C01814=1073.013,225.555,417.556,174.109,27.687,154.920
C01815=1073.019,225.804,417.531,174.111,27.690,154.921
C01816=1073.025,226.052,417.504,174.113,27.694,154.921
C01817=1073.031,226.301,417.478,174.116,27.698,154.922
C01818=1073.036,226.549,417.451,174.118,27.702,154.923
C01819=1073.043,226.798,417.426,174.120,27.706,154.923
C01820=1073.048,227.046,417.399,174.123,27.710,154.924
C01821=1073.054,227.295,417.373,174.125,27.713,154.924
C01822=1073.060,227.544,417.348,174.127,27.717,154.925
C01823=1073.066,227.792,417.321,174.129,27.721,154.926
C01824=1073.072,228.041,417.295,174.131,27.725,154.926
C01825=1073.078,228.289,417.269,174.133,27.729,154.927
C01826=1073.084,228.538,417.243,174.136,27.733,154.927
C01827=1073.089,228.787,417.217,174.138,27.736,154.928
C01828=1073.096,229.036,417.190,174.140,27.740,154.929
C01829=1073.102,229.285,417.165,174.143,27.744,154.929
C01830=1073.107,229.533,417.138,174.145,27.748,154.930
C01831=1073.113,229.782,417.112,174.147,27.752,154.930
C01832=1073.119,230.030,417.086,174.150,27.755,154.931
C01833=1073.125,230.278,417.059,174.152,27.760,154.932
C01834=1073.131,230.527,417.033,174.154,27.764,154.932
C01835=1073.136,230.776,417.007,174.156,27.768,154.933
C01836=1073.142,231.024,416.980,174.158,27.771,154.933
C01837=1073.148,231.273,416.954,174.160,27.775,154.934
C01838=1073.153,231.521,416.927,174.163,27.779,154.935
C01839=1073.159,231.770,416.901,174.165,27.782,154.935
C01840=1073.165,232.018,416.874,174.167,27.787,154.936
C01841=1073.170,232.267,416.848,174.169,27.791,154.936
C01842=1073.177,232.515,416.822,174.172,27.795,154.937
C01843=1073.183,232.764,416.795,174.174,27.798,154.938
C01844=1073.189,233.013,416.769,174.176,27.802,154.938
C01845=1073.195,233.262,416.743,174.179,27.806,154.939
C01846=1073.200,233.510,416.716,174.181,27.810,154.939
C01847=1073.206,233.758,416.689,174.183,27.814,154.940
C01848=1073.212,234.007,416.663,174.186,27.818,154.941
C01849=1073.218,234.255,416.636,174.188,27.821,154.941
C01850=1073.223,234.504,416.610,174.190,27.825,154.942
C01851=1073.229,234.752,416.583,174.193,27.829,154.943
C01852=1073.235,235.001,416.557,174.195,27.833,154.943
C01853=1073.244,235.416,416.511,174.198,27.839,154.944
C01854=1073.254,235.831,416.467,174.202,27.846,154.945
C01855=1073.264,236.245,416.423,174.206,27.852,154.946
C01856=1073.273,236.660,416.377,174.210,27.859,154.947
C01857=1073.279,236.908,416.351,174.212,27.863,154.948
C01858=1073.285,237.157,416.324,174.214,27.867,154.948
C01859=1073.291,237.405,416.297,174.217,27.871,154.949
C01860=1073.296,237.653,416.271,174.219,27.874,154.950
C01861=1073.303,237.902,416.244,174.221,27.878,154.950
C01862=1073.309,238.151,416.217,174.224,27.882,154.951
C01863=1073.314,238.399,416.191,174.226,27.886,154.951
C01864=1073.320,238.648,416.164,174.228,27.890,154.952
C01865=1073.327,238.897,416.137,174.231,27.894,154.953
C01866=1073.332,239.145,416.110,174.233,27.897,154.953
C01867=1073.337,239.394,416.083,174.235,27.901,154.954
C01868=1073.343,239.642,416.056,174.238,27.905,154.954
C01869=1073.350,239.891,416.029,174.240,27.909,154.955
C01870=1073.355,240.139,416.003,174.242,27.913,154.956
C01871=1073.361,240.387,415.975,174.245,27.917,154.956
C01872=1073.367,240.636,415.949,174.247,27.920,154.957
C01873=1073.373,240.885,415.921,174.249,27.924,154.957
C01874=1073.379,241.133,415.894,174.252,27.928,154.958
C01875=1073.384,241.382,415.868,174.254,27.932,154.959
C01876=1073.390,241.629,415.840,174.257,27.936,154.959
C01877=1073.397,241.878,415.813,174.259,27.940,154.960
C01878=1073.402,242.127,415.786,174.261,27.943,154.960
C01879=1073.408,242.375,415.759,174.264,27.947,154.961
C01880=1073.414,242.624,415.732,174.266,27.951,154.962
C01881=1073.420,242.872,415.705,174.268,27.955,154.962
C01882=1073.425,243.121,415.678,174.271,27.959,154.963
C01883=1073.431,243.369,415.650,174.273,27.963,154.963
C01884=1073.438,243.618,415.623,174.275,27.967,154.964
C01885=1073.443,243.866,415.596,174.278,27.971,154.965
C01886=1073.449,244.114,415.569,174.280,27.975,154.965
C01887=1073.454,244.364,415.541,174.282,27.978,154.966
C01888=1073.460,244.612,415.515,174.285,27.982,154.966
C01889=1073.466,244.860,415.487,174.287,27.986,154.967
C01890=1073.472,245.109,415.460,174.289,27.990,154.968
C01891=1073.478,245.357,415.432,174.292,27.994,154.968
C01892=1073.483,245.605,415.405,174.294,27.998,154.969
C01893=1073.490,245.854,415.377,174.296,28.002,154.970
C01894=1073.495,246.103,415.350,174.300,28.005,154.970
C01895=1073.500,246.351,415.323,174.302,28.009,154.971
C01896=1073.507,246.599,415.296,174.304,28.013,154.971
C01897=1073.512,246.848,415.268,174.307,28.017,154.972
C01898=1073.518,247.096,415.241,174.309,28.021,154.972
C01899=1073.524,247.344,415.213,174.312,28.025,154.973
C01900=1073.529,247.593,415.185,174.314,28.029,154.974
C01901=1073.535,247.841,415.158,174.316,28.033,154.974
C01902=1073.541,248.090,415.131,174.319,28.036,154.975
C01903=1073.547,248.338,415.103,174.321,28.040,154.976
C01904=1073.552,248.587,415.076,174.323,28.045,154.976
C01905=1073.562,248.995,415.030,174.327,28.051,154.977
C01906=1073.571,249.403,414.985,174.331,28.057,154.978
C01907=1073.581,249.812,414.939,174.335,28.064,154.979
C01908=1073.590,250.219,414.893,174.339,28.070,154.980
C01909=1073.595,250.468,414.866,174.341,28.074,154.981
C01910=1073.601,250.716,414.839,174.344,28.078,154.982
C01911=1073.607,250.965,414.810,174.346,28.082,154.982
C01912=1073.613,251.213,414.782,174.348,28.086,154.983
C01913=1073.619,251.462,414.755,174.351,28.090,154.983
C01914=1073.624,251.710,414.727,174.353,28.094,154.984
C01915=1073.630,251.958,414.699,174.356,28.097,154.985
C01916=1073.636,252.206,414.672,174.359,28.101,154.985
C01917=1073.641,252.455,414.644,174.361,28.105,154.986
C01918=1073.647,252.704,414.616,174.363,28.109,154.986
C01919=1073.653,252.951,414.589,174.366,28.113,154.987
C01920=1073.659,253.200,414.560,174.368,28.117,154.988
C01921=1073.665,253.448,414.532,174.371,28.121,154.988
C01922=1073.671,253.697,414.505,174.373,28.125,154.989
C01923=1073.677,253.945,414.477,174.375,28.128,154.989
C01924=1073.683,254.193,414.448,174.378,28.132,154.990
C01925=1073.688,254.442,414.421,174.380,28.136,154.991
C01926=1073.694,254.691,414.393,174.383,28.140,154.991
C01927=1073.700,254.939,414.365,174.386,28.144,154.992
C01928=1073.706,255.187,414.337,174.388,28.148,154.993
C01929=1073.712,255.436,414.309,174.390,28.152,154.993
C01930=1073.718,255.684,414.281,174.393,28.156,154.994
C01931=1073.724,255.933,414.253,174.395,28.160,154.994
C01932=1073.729,256.181,414.225,174.398,28.164,154.995
C01933=1073.735,256.429,414.197,174.400,28.167,154.996
C01934=1073.741,256.677,414.169,174.402,28.171,154.996
C01935=1073.747,256.926,414.141,174.406,28.175,154.997
C01936=1073.753,257.175,414.113,174.408,28.179,154.997
C01937=1073.758,257.423,414.085,174.410,28.183,154.998
C01938=1073.765,257.671,414.056,174.413,28.187,154.999
C01939=1073.771,257.919,414.028,174.415,28.190,154.999
C01940=1073.776,258.167,414.000,174.418,28.194,155.000
C01941=1073.782,258.416,413.972,174.420,28.198,155.000
C01942=1073.788,258.664,413.944,174.422,28.202,155.001
C01943=1073.794,258.913,413.916,174.426,28.206,155.002
C01944=1073.800,259.161,413.888,174.428,28.210,155.002
C01945=1073.806,259.409,413.859,174.430,28.214,155.003
C01946=1073.812,259.657,413.831,174.433,28.217,155.003
C01947=1073.818,259.906,413.802,174.435,28.221,155.004
C01948=1073.824,260.154,413.775,174.438,28.225,155.005
C01949=1073.830,260.403,413.747,174.440,28.229,155.005
C01950=1073.836,260.651,413.718,174.443,28.233,155.006
C01951=1073.842,260.899,413.690,174.446,28.237,155.006
C01952=1073.847,261.148,413.661,174.448,28.241,155.007
C01953=1073.854,261.396,413.632,174.450,28.245,155.008
C01954=1073.860,261.644,413.605,174.453,28.248,155.008
C01955=1073.866,261.892,413.577,174.455,28.252,155.009
C01956=1073.872,262.140,413.548,174.459,28.256,155.009
C01957=1073.881,262.547,413.501,174.463,28.262,155.010
C01958=1073.891,262.952,413.455,174.467,28.268,155.011
C01959=1073.902,263.357,413.409,174.471,28.275,155.012
C01960=1073.911,263.764,413.362,174.475,28.281,155.013
C01961=1073.917,264.011,413.334,174.477,28.285,155.014
C01962=1073.923,264.260,413.305,174.480,28.289,155.015
C01963=1073.929,264.508,413.276,174.483,28.293,155.015
C01964=1073.934,264.756,413.248,174.485,28.297,155.016
C01965=1073.941,265.004,413.219,174.488,28.300,155.016
C01966=1073.946,265.253,413.190,174.490,28.304,155.017
C01967=1073.952,265.502,413.161,174.493,28.309,155.018
C01968=1073.957,265.750,413.133,174.496,28.312,155.018
C01969=1073.964,265.998,413.104,174.498,28.316,155.019
C01970=1073.970,266.246,413.075,174.500,28.320,155.019
C01971=1073.976,266.495,413.047,174.503,28.324,155.020
C01972=1073.981,266.742,413.018,174.505,28.328,155.021
C01973=1073.987,266.991,412.989,174.508,28.332,155.021
C01974=1073.993,267.239,412.960,174.511,28.336,155.022
C01975=1073.999,267.487,412.931,174.513,28.340,155.023
C01976=1074.005,267.736,412.903,174.516,28.343,155.023
C01977=1074.010,267.984,412.874,174.518,28.347,155.024
C01978=1074.016,268.232,412.845,174.521,28.352,155.025
C01979=1074.022,268.481,412.816,174.524,28.355,155.025
C01980=1074.028,268.729,412.787,174.526,28.359,155.026
C01981=1074.035,268.977,412.758,174.529,28.363,155.026
C01982=1074.040,269.226,412.728,174.532,28.367,155.027
C01983=1074.046,269.474,412.701,174.534,28.371,155.028
C01984=1074.052,269.722,412.671,174.537,28.375,155.028
C01985=1074.057,269.970,412.642,174.539,28.379,155.029
C01986=1074.064,270.218,412.613,174.542,28.383,155.029
C01987=1074.070,270.466,412.584,174.545,28.387,155.030
C01988=1074.076,270.715,412.555,174.547,28.391,155.031
C01989=1074.081,270.963,412.526,174.550,28.395,155.031
C01990=1074.087,271.211,412.497,174.552,28.399,155.032
C01991=1074.092,271.459,412.467,174.555,28.402,155.033
C01992=1074.099,271.708,412.438,174.558,28.406,155.033
C01993=1074.105,271.956,412.409,174.560,28.410,155.034
C01994=1074.110,272.204,412.380,174.563,28.414,155.034
C01995=1074.117,272.452,412.351,174.565,28.418,155.035
C01996=1074.123,272.700,412.322,174.568,28.423,155.036
C01997=1074.128,272.949,412.292,174.571,28.426,155.036
C01998=1074.134,273.196,412.263,174.573,28.430,155.037
C01999=1074.140,273.445,412.234,174.576,28.434,155.038
C02000=1074.146,273.693,412.205,174.579,28.438,155.038
C02001=1074.151,273.941,412.175,174.581,28.442,155.039
C02002=1074.158,274.189,412.146,174.584,28.446,155.040
C02003=1074.163,274.438,412.116,174.586,28.450,155.040
C02004=1074.169,274.686,412.087,174.589,28.454,155.041
C02005=1074.175,274.934,412.058,174.592,28.458,155.041
C02006=1074.181,275.183,412.029,174.594,28.462,155.042
C02007=1074.187,275.431,411.999,174.597,28.466,155.043
C02008=1074.193,275.679,411.970,174.600,28.470,155.043
C02009=1074.202,276.088,411.922,174.604,28.476,155.044
C02010=1074.212,276.496,411.872,174.609,28.483,155.045
C02011=1074.222,276.906,411.824,174.613,28.489,155.046
C02012=1074.232,277.314,411.776,174.617,28.496,155.047
C02013=1074.237,277.562,411.746,174.620,28.500,155.048
C02014=1074.243,277.811,411.717,174.623,28.504,155.049
C02015=1074.249,278.058,411.687,174.625,28.508,155.049
C02016=1074.255,278.307,411.657,174.627,28.512,155.050
C02017=1074.261,278.555,411.628,174.631,28.516,155.051
C02018=1074.267,278.803,411.598,174.633,28.520,155.051
C02019=1074.272,279.051,411.568,174.636,28.524,155.052
C02020=1074.279,279.299,411.539,174.639,28.528,155.052
C02021=1074.284,279.547,411.509,174.641,28.532,155.053
C02022=1074.290,279.796,411.479,174.644,28.536,155.054
C02023=1074.296,280.044,411.450,174.646,28.540,155.054
C02024=1074.303,280.292,411.419,174.650,28.544,155.055
C02025=1074.308,280.541,411.390,174.652,28.548,155.056
C02026=1074.315,280.788,411.360,174.654,28.552,155.056
C02027=1074.320,281.037,411.330,174.658,28.556,155.057
C02028=1074.326,281.285,411.301,174.660,28.560,155.058
C02029=1074.332,281.533,411.270,174.663,28.564,155.058
C02030=1074.337,281.781,411.241,174.666,28.568,155.059
C02031=1074.344,282.029,411.211,174.668,28.572,155.060
C02032=1074.349,282.277,411.181,174.671,28.576,155.060
C02033=1074.355,282.525,411.151,174.674,28.580,155.061
C02034=1074.361,282.773,411.121,174.676,28.584,155.062
C02035=1074.366,283.021,411.091,174.679,28.588,155.062
C02036=1074.372,283.269,411.061,174.681,28.592,155.063
C02037=1074.378,283.517,411.032,174.685,28.596,155.063
C02038=1074.385,283.766,411.001,174.687,28.600,155.064
C02039=1074.391,284.014,410.971,174.689,28.605,155.065
C02040=1074.396,284.262,410.941,174.693,28.609,155.066
C02041=1074.402,284.510,410.911,174.695,28.613,155.066
C02042=1074.407,284.758,410.881,174.698,28.617,155.067
C02043=1074.413,285.006,410.851,174.701,28.621,155.067
C02044=1074.419,285.254,410.820,174.703,28.625,155.068
C02045=1074.426,285.502,410.790,174.707,28.629,155.069
C02046=1074.432,285.751,410.760,174.709,28.633,155.069
C02047=1074.438,285.999,410.730,174.712,28.637,155.070
C02048=1074.443,286.246,410.700,174.715,28.641,155.071
C02049=1074.449,286.494,410.669,174.717,28.645,155.071
C02050=1074.455,286.743,410.639,174.720,28.649,155.072
C02051=1074.461,286.991,410.609,174.723,28.653,155.073
C02052=1074.467,287.239,410.579,174.726,28.657,155.073
C02053=1074.473,287.487,410.548,174.728,28.661,155.074
C02054=1074.479,287.735,410.518,174.731,28.665,155.075
C02055=1074.485,287.984,410.488,174.734,28.669,155.075
C02056=1074.491,288.231,410.458,174.736,28.673,155.076
C02057=1074.497,288.479,410.428,174.740,28.677,155.077
C02058=1074.503,288.727,410.398,174.742,28.681,155.077
C02059=1074.509,288.975,410.367,174.745,28.685,155.078
C02060=1074.515,289.223,410.336,174.748,28.689,155.078
C02061=1074.525,289.642,410.285,174.753,28.696,155.080
C02062=1074.535,290.061,410.234,174.757,28.703,155.081
C02063=1074.545,290.480,410.182,174.762,28.710,155.082
C02064=1074.555,290.899,410.131,174.767,28.717,155.083
C02065=1074.560,291.147,410.100,174.769,28.721,155.084
C02066=1074.566,291.396,410.069,174.772,28.725,155.084
C02067=1074.572,291.643,410.039,174.775,28.729,155.085
C02068=1074.578,291.891,410.008,174.777,28.734,155.086
C02069=1074.585,292.139,409.977,174.781,28.738,155.086
C02070=1074.591,292.387,409.947,174.783,28.742,155.087
C02071=1074.596,292.635,409.916,174.786,28.746,155.088
C02072=1074.602,292.883,409.885,174.789,28.750,155.088
C02073=1074.608,293.131,409.855,174.791,28.754,155.089
C02074=1074.614,293.379,409.824,174.795,28.758,155.090
C02075=1074.620,293.626,409.793,174.797,28.762,155.090
C02076=1074.626,293.875,409.762,174.800,28.766,155.091
C02077=1074.631,294.123,409.732,174.803,28.770,155.092
C02078=1074.638,294.372,409.701,174.806,28.775,155.092
C02079=1074.644,294.619,409.670,174.809,28.779,155.093
C02080=1074.650,294.867,409.639,174.811,28.783,155.094
C02081=1074.655,295.115,409.608,174.814,28.787,155.094
C02082=1074.662,295.363,409.577,174.817,28.792,155.095
C02083=1074.667,295.610,409.547,174.820,28.796,155.096
C02084=1074.673,295.859,409.515,174.823,28.800,155.096
C02085=1074.679,296.107,409.484,174.826,28.804,155.097
C02086=1074.686,296.355,409.454,174.828,28.808,155.098
C02087=1074.691,296.603,409.423,174.831,28.812,155.099
C02088=1074.697,296.850,409.392,174.834,28.816,155.099
C02089=1074.703,297.099,409.361,174.837,28.820,155.100
C02090=1074.709,297.346,409.329,174.840,28.825,155.101
C02091=1074.715,297.595,409.298,174.842,28.829,155.101
C02092=1074.720,297.842,409.267,174.846,28.833,155.102
C02093=1074.727,298.091,409.236,174.848,28.837,155.103
C02094=1074.732,298.339,409.204,174.852,28.842,155.103
C02095=1074.738,298.586,409.174,174.854,28.846,155.104
C02096=1074.744,298.835,409.142,174.857,28.850,155.105
C02097=1074.750,299.082,409.112,174.860,28.855,155.106
C02098=1074.755,299.330,409.080,174.862,28.858,155.106
C02099=1074.761,299.579,409.049,174.866,28.863,155.107
C02100=1074.767,299.826,409.018,174.868,28.867,155.108
C02101=1074.773,300.074,408.986,174.871,28.872,155.108
C02102=1074.779,300.322,408.955,174.874,28.876,155.109
C02103=1074.785,300.570,408.923,174.877,28.880,155.110
C02104=1074.790,300.818,408.892,174.880,28.884,155.110
C02105=1074.796,301.065,408.861,174.883,28.889,155.111
C02106=1074.802,301.314,408.829,174.885,28.893,155.112
C02107=1074.807,301.561,408.798,174.889,28.897,155.113
C02108=1074.814,301.810,408.767,174.891,28.901,155.113
C02109=1074.819,302.057,408.735,174.894,28.906,155.114
C02110=1074.825,302.305,408.703,174.897,28.910,155.115
C02111=1074.831,302.553,408.672,174.900,28.915,155.115
C02112=1074.837,302.801,408.640,174.903,28.918,155.116
C02113=1074.842,303.017,408.613,174.905,28.922,155.117
C02114=1074.847,303.235,408.585,174.908,28.926,155.117
C02115=1074.852,303.451,408.558,174.910,28.930,155.118
C02116=1074.858,303.668,408.530,174.913,28.934,155.119
C02117=1074.863,303.885,408.503,174.916,28.938,155.119
C02118=1074.868,304.102,408.475,174.919,28.941,155.120
C02119=1074.873,304.318,408.447,174.921,28.945,155.120
C02120=1074.879,304.535,408.420,174.923,28.949,155.121
C02121=1074.884,304.783,408.388,174.926,28.953,155.122
C02122=1074.890,305.031,408.356,174.929,28.957,155.123
C02123=1074.897,305.279,408.325,174.932,28.961,155.123
C02124=1074.902,305.526,408.293,174.935,28.966,155.124
C02125=1074.908,305.775,408.261,174.938,28.970,155.125
C02126=1074.914,306.022,408.230,174.941,28.975,155.125
C02127=1074.920,306.270,408.198,174.943,28.979,155.126
C02128=1074.926,306.518,408.166,174.947,28.983,155.127
C02129=1074.932,306.766,408.134,174.950,28.988,155.128
C02130=1074.938,307.014,408.103,174.952,28.992,155.128
C02131=1074.944,307.262,408.071,174.956,28.996,155.129
C02132=1074.950,307.509,408.039,174.958,29.000,155.130
C02133=1074.956,307.758,408.007,174.962,29.005,155.130
C02134=1074.962,308.005,407.976,174.964,29.009,155.131
C02135=1074.968,308.252,407.943,174.967,29.013,155.132
C02136=1074.974,308.501,407.911,174.970,29.018,155.133
C02137=1074.980,308.749,407.879,174.973,29.022,155.133
C02138=1074.986,308.996,407.848,174.977,29.027,155.134
C02139=1074.992,309.244,407.816,174.979,29.030,155.135
C02140=1074.998,309.492,407.784,174.982,29.035,155.136
C02141=1075.004,309.740,407.751,174.985,29.039,155.136
C02142=1075.011,309.987,407.720,174.988,29.044,155.137
C02143=1075.017,310.235,407.688,174.991,29.048,155.138
C02144=1075.023,310.484,407.656,174.994,29.052,155.138
C02145=1075.029,310.731,407.623,174.998,29.057,155.139
C02146=1075.035,310.979,407.591,175.000,29.061,155.140
C02147=1075.040,311.227,407.560,175.003,29.065,155.141
C02148=1075.047,311.474,407.528,175.006,29.070,155.141
C02149=1075.053,311.722,407.496,175.009,29.074,155.142
C02150=1075.059,311.971,407.464,175.013,29.078,155.143
C02151=1075.066,312.218,407.431,175.015,29.083,155.144
C02152=1075.072,312.466,407.399,175.018,29.087,155.144
C02153=1075.077,312.714,407.367,175.021,29.091,155.145
C02154=1075.084,312.961,407.335,175.024,29.096,155.146
C02155=1075.090,313.209,407.303,175.028,29.100,155.146
C02156=1075.096,313.457,407.270,175.030,29.104,155.147
C02157=1075.102,313.705,407.238,175.033,29.109,155.148
C02158=1075.109,313.953,407.205,175.036,29.113,155.149
C02159=1075.115,314.201,407.173,175.039,29.118,155.149
C02160=1075.121,314.449,407.141,175.043,29.122,155.150
C02161=1075.127,314.697,407.109,175.045,29.127,155.151
C02162=1075.132,314.944,407.076,175.048,29.131,155.152
C02163=1075.138,315.192,407.044,175.051,29.136,155.152
C02164=1075.144,315.440,407.011,175.054,29.140,155.153
C02165=1075.150,315.687,406.978,175.058,29.145,155.154
C02166=1075.156,315.936,406.946,175.060,29.149,155.155
C02167=1075.161,316.183,406.913,175.063,29.154,155.156
C02168=1075.168,316.431,406.880,175.066,29.158,155.156
C02169=1075.174,316.681,406.848,175.069,29.163,155.157
C02170=1075.180,316.930,406.815,175.073,29.168,155.158
C02171=1075.185,317.180,406.782,175.075,29.172,155.159
C02172=1075.191,317.429,406.750,175.078,29.177,155.159
C02173=1075.197,317.677,406.717,175.082,29.181,155.160
C02174=1075.203,317.925,406.683,175.084,29.186,155.161
C02175=1075.209,318.173,406.651,175.088,29.190,155.162
C02176=1075.215,318.420,406.618,175.091,29.195,155.163
C02177=1075.221,318.669,406.585,175.093,29.199,155.163
C02178=1075.227,318.916,406.553,175.097,29.204,155.164
C02179=1075.233,319.164,406.520,175.100,29.209,155.165
C02180=1075.239,319.412,406.487,175.103,29.213,155.166
C02181=1075.245,319.659,406.454,175.106,29.218,155.167
C02182=1075.251,319.907,406.420,175.108,29.222,155.167
C02183=1075.257,320.155,406.388,175.112,29.227,155.168
C02184=1075.263,320.403,406.356,175.115,29.232,155.169
C02185=1075.268,320.651,406.322,175.118,29.236,155.170
C02186=1075.275,320.899,406.290,175.121,29.241,155.170
C02187=1075.280,321.146,406.256,175.124,29.246,155.171
C02188=1075.287,321.394,406.224,175.127,29.250,155.172
C02189=1075.292,321.611,406.195,175.130,29.254,155.173
C02190=1075.297,321.829,406.165,175.133,29.258,155.173
C02191=1075.302,322.046,406.137,175.135,29.262,155.174
C02192=1075.308,322.263,406.107,175.138,29.266,155.175
C02193=1075.313,322.480,406.079,175.141,29.270,155.175
C02194=1075.318,322.698,406.049,175.144,29.274,155.176
C02195=1075.324,322.916,406.020,175.146,29.279,155.177
C02196=1075.329,323.133,405.991,175.149,29.282,155.178
C02197=1075.335,323.380,405.959,175.152,29.287,155.178
C02198=1075.341,323.628,405.925,175.155,29.292,155.179
C02199=1075.347,323.876,405.893,175.158,29.297,155.180
C02200=1075.353,324.125,405.859,175.161,29.301,155.181
C02201=1075.360,324.372,405.825,175.165,29.306,155.182
C02202=1075.365,324.619,405.792,175.168,29.310,155.182
C02203=1075.371,324.867,405.759,175.170,29.315,155.183
C02204=1075.377,325.115,405.726,175.174,29.320,155.184
C02205=1075.383,325.363,405.693,175.177,29.324,155.185
C02206=1075.390,325.611,405.659,175.180,29.329,155.186
C02207=1075.396,325.858,405.626,175.183,29.334,155.187
C02208=1075.402,326.106,405.593,175.186,29.339,155.187
C02209=1075.408,326.353,405.559,175.190,29.343,155.188
C02210=1075.414,326.601,405.526,175.192,29.347,155.189
C02211=1075.421,326.849,405.493,175.196,29.353,155.190
C02212=1075.426,327.096,405.459,175.199,29.357,155.191
C02213=1075.433,327.344,405.426,175.202,29.362,155.191
C02214=1075.438,327.592,405.393,175.205,29.367,155.192
C02215=1075.446,327.840,405.359,175.208,29.371,155.193
C02216=1075.451,328.088,405.325,175.212,29.376,155.194
C02217=1075.458,328.335,405.292,175.215,29.381,155.195
C02218=1075.463,328.582,405.259,175.217,29.385,155.195
C02219=1075.470,328.830,405.224,175.221,29.390,155.196
C02220=1075.476,329.078,405.192,175.224,29.395,155.197
C02221=1075.482,329.325,405.157,175.228,29.400,155.198
C02222=1075.489,329.574,405.124,175.231,29.404,155.199
C02223=1075.495,329.821,405.090,175.233,29.409,155.200
C02224=1075.501,330.068,405.058,175.237,29.414,155.200
C02225=1075.506,330.283,405.028,175.239,29.418,155.201
C02226=1075.512,330.500,404.999,175.243,29.422,155.202
C02227=1075.518,330.714,404.969,175.245,29.426,155.203
C02228=1075.522,330.930,404.940,175.248,29.430,155.203
C02229=1075.528,331.145,404.911,175.251,29.434,155.204
C02230=1075.534,331.359,404.882,175.254,29.439,155.205
C02231=1075.538,331.575,404.852,175.256,29.443,155.206
C02232=1075.543,331.790,404.822,175.259,29.447,155.206
C02233=1075.551,332.038,404.789,175.262,29.452,155.207
C02234=1075.556,332.286,404.755,175.265,29.457,155.208
C02235=1075.562,332.533,404.721,175.269,29.462,155.209
C02236=1075.568,332.781,404.687,175.272,29.467,155.210
C02237=1075.574,333.028,404.653,175.275,29.472,155.211
C02238=1075.580,333.276,404.619,175.278,29.476,155.211
C02239=1075.586,333.524,404.585,175.281,29.481,155.212
C02240=1075.592,333.771,404.551,175.285,29.486,155.213
C02241=1075.598,334.019,404.517,175.288,29.491,155.214
C02242=1075.605,334.267,404.482,175.292,29.496,155.215
C02243=1075.610,334.514,404.448,175.294,29.501,155.216
C02244=1075.616,334.761,404.414,175.297,29.506,155.217
C02245=1075.622,335.010,404.381,175.301,29.511,155.218
C02246=1075.628,335.257,404.347,175.304,29.516,155.218
C02247=1075.635,335.505,404.313,175.308,29.521,155.219
C02248=1075.641,335.752,404.279,175.311,29.526,155.220
C02249=1075.648,336.000,404.244,175.313,29.531,155.221
C02250=1075.654,336.247,404.210,175.317,29.536,155.222
C02251=1075.660,336.495,404.176,175.320,29.541,155.223
C02252=1075.666,336.743,404.142,175.324,29.546,155.224
C02253=1075.672,336.991,404.107,175.327,29.550,155.224
C02254=1075.679,337.237,404.073,175.330,29.556,155.225
C02255=1075.685,337.485,404.038,175.334,29.561,155.226
C02256=1075.691,337.732,404.004,175.336,29.565,155.227
C02257=1075.697,337.980,403.970,175.340,29.571,155.228
C02258=1075.703,338.228,403.935,175.343,29.576,155.229
C02259=1075.708,338.475,403.901,175.346,29.581,155.230
C02260=1075.715,338.723,403.867,175.350,29.586,155.231
C02261=1075.721,338.970,403.832,175.353,29.591,155.232
C02262=1075.727,339.218,403.797,175.357,29.596,155.233
C02263=1075.733,339.466,403.763,175.360,29.601,155.233
C02264=1075.739,339.714,403.728,175.362,29.606,155.234
C02265=1075.745,339.960,403.694,175.366,29.611,155.235
C02266=1075.752,340.208,403.659,175.369,29.616,155.236
C02267=1075.758,340.456,403.625,175.373,29.622,155.237
C02268=1075.764,340.703,403.589,175.376,29.627,155.238
C02269=1075.770,340.951,403.555,175.379,29.632,155.239
C02270=1075.776,341.198,403.521,175.383,29.637,155.240
C02271=1075.783,341.446,403.486,175.386,29.642,155.241
C02272=1075.788,341.693,403.451,175.390,29.647,155.242
C02273=1075.795,341.941,403.416,175.393,29.652,155.243
C02274=1075.801,342.189,403.382,175.396,29.658,155.244
C02275=1075.807,342.436,403.348,175.399,29.662,155.245
C02276=1075.813,342.684,403.312,175.402,29.668,155.246
C02277=1075.819,342.932,403.277,175.406,29.673,155.247
C02278=1075.826,343.178,403.243,175.409,29.678,155.247
C02279=1075.832,343.426,403.208,175.412,29.683,155.248
C02280=1075.838,343.674,403.172,175.416,29.689,155.249
C02281=1075.843,343.886,403.142,175.419,29.693,155.250
C02282=1075.849,344.099,403.113,175.422,29.698,155.251
C02283=1075.854,344.311,403.083,175.424,29.702,155.252
C02284=1075.859,344.524,403.053,175.428,29.706,155.253
C02285=1075.865,344.736,403.022,175.430,29.711,155.253
C02286=1075.869,344.949,402.993,175.434,29.716,155.254
C02287=1075.875,345.162,402.963,175.436,29.720,155.255
C02288=1075.880,345.374,402.933,175.439,29.724,155.256
C02289=1075.886,345.621,402.897,175.442,29.730,155.257
C02290=1075.893,345.869,402.863,175.445,29.735,155.258
C02291=1075.899,346.116,402.828,175.449,29.741,155.259
C02292=1075.905,346.364,402.792,175.452,29.746,155.260
C02293=1075.912,346.611,402.757,175.456,29.751,155.261
C02294=1075.917,346.858,402.722,175.459,29.757,155.262
C02295=1075.923,347.106,402.687,175.462,29.762,155.263
C02296=1075.930,347.354,402.651,175.466,29.767,155.264
C02297=1075.936,347.601,402.616,175.469,29.772,155.265
C02298=1075.942,347.848,402.581,175.473,29.778,155.266
C02299=1075.948,348.096,402.545,175.476,29.783,155.267
C02300=1075.955,348.343,402.510,175.479,29.789,155.268
C02301=1075.961,348.591,402.474,175.483,29.794,155.269
C02302=1075.968,348.838,402.439,175.486,29.800,155.270
C02303=1075.973,349.085,402.404,175.490,29.805,155.270
C02304=1075.979,349.333,402.368,175.493,29.810,155.272
C02305=1075.986,349.580,402.333,175.496,29.816,155.273
C02306=1075.992,349.828,402.297,175.500,29.821,155.274
C02307=1075.999,350.075,402.262,175.503,29.826,155.274
C02308=1076.004,350.322,402.227,175.507,29.832,155.276
C02309=1076.010,350.570,402.191,175.510,29.837,155.277
C02310=1076.017,350.817,402.156,175.513,29.843,155.278
C02311=1076.023,351.065,402.120,175.517,29.849,155.279
C02312=1076.030,351.312,402.085,175.520,29.854,155.280
C02313=1076.036,351.560,402.049,175.524,29.859,155.281
C02314=1076.042,351.807,402.013,175.528,29.865,155.282
C02315=1076.048,352.054,401.978,175.531,29.870,155.283
C02316=1076.054,352.301,401.942,175.535,29.876,155.284
C02317=1076.060,352.549,401.907,175.538,29.881,155.285
C02318=1076.066,352.797,401.871,175.542,29.887,155.286
C02319=1076.073,353.043,401.835,175.545,29.893,155.287
C02320=1076.079,353.291,401.799,175.548,29.898,155.288
C02321=1076.085,353.539,401.764,175.552,29.904,155.289
C02322=1076.092,353.786,401.727,175.555,29.909,155.290
C02323=1076.098,354.033,401.691,175.559,29.915,155.291
C02324=1076.104,354.281,401.656,175.562,29.921,155.292
C02325=1076.110,354.527,401.620,175.565,29.926,155.293
C02326=1076.116,354.775,401.584,175.569,29.932,155.294
C02327=1076.123,355.022,401.548,175.572,29.937,155.295
C02328=1076.129,355.270,401.512,175.576,29.943,155.296
C02329=1076.135,355.517,401.476,175.580,29.949,155.297
C02330=1076.141,355.764,401.440,175.583,29.955,155.298
C02331=1076.147,356.011,401.404,175.587,29.960,155.299
C02332=1076.153,356.259,401.368,175.590,29.966,155.300
C02333=1076.160,356.506,401.332,175.593,29.972,155.302
C02334=1076.166,356.753,401.296,175.597,29.977,155.303
C02335=1076.173,357.001,401.260,175.600,29.983,155.304
C02336=1076.179,357.248,401.223,175.604,29.989,155.305
C02337=1076.185,357.463,401.192,175.607,29.994,155.306
C02338=1076.190,357.677,401.161,175.611,29.999,155.307
C02339=1076.195,357.891,401.129,175.613,30.004,155.307
C02340=1076.201,358.105,401.099,175.617,30.009,155.308
C02341=1076.207,358.319,401.067,175.619,30.013,155.309
C02342=1076.212,358.534,401.035,175.623,30.018,155.310
C02343=1076.217,358.747,401.004,175.626,30.024,155.311
C02344=1076.223,358.962,400.973,175.628,30.029,155.312
C02345=1076.230,359.209,400.936,175.632,30.034,155.313
C02346=1076.236,359.457,400.900,175.635,30.040,155.314
C02347=1076.242,359.704,400.863,175.640,30.046,155.315
C02348=1076.248,359.951,400.828,175.643,30.052,155.317
C02349=1076.255,360.198,400.791,175.646,30.058,155.318
C02350=1076.260,360.446,400.754,175.650,30.063,155.319
C02351=1076.267,360.693,400.718,175.653,30.070,155.320
C02352=1076.273,360.940,400.681,175.657,30.076,155.321
C02353=1076.279,361.187,400.645,175.661,30.081,155.322
C02354=1076.286,361.434,400.608,175.664,30.087,155.323
C02355=1076.293,361.682,400.571,175.668,30.093,155.324
C02356=1076.299,361.929,400.535,175.671,30.099,155.326
C02357=1076.305,362.176,400.499,175.675,30.105,155.327
C02358=1076.311,362.423,400.462,175.679,30.111,155.328
C02359=1076.317,362.670,400.425,175.682,30.117,155.329
C02360=1076.324,362.918,400.388,175.686,30.123,155.330
C02361=1076.330,363.165,400.352,175.689,30.129,155.331
C02362=1076.337,363.412,400.315,175.693,30.135,155.332
C02363=1076.343,363.659,400.278,175.697,30.141,155.334
C02364=1076.349,363.906,400.241,175.700,30.147,155.335
C02365=1076.356,364.154,400.204,175.704,30.153,155.336
C02366=1076.362,364.401,400.168,175.707,30.159,155.337
C02367=1076.369,364.648,400.131,175.711,30.165,155.338
C02368=1076.375,364.894,400.094,175.715,30.172,155.339
C02369=1076.381,365.142,400.057,175.718,30.178,155.341
C02370=1076.388,365.389,400.020,175.722,30.184,155.342
C02371=1076.393,365.637,399.983,175.725,30.190,155.343
C02372=1076.400,365.883,399.946,175.730,30.196,155.344
C02373=1076.406,366.131,399.909,175.733,30.202,155.345
C02374=1076.413,366.378,399.872,175.736,30.208,155.346
C02375=1076.418,366.625,399.835,175.740,30.214,155.348
C02376=1076.425,366.872,399.798,175.744,30.220,155.349
C02377=1076.432,367.119,399.761,175.748,30.227,155.350
C02378=1076.438,367.366,399.724,175.751,30.233,155.351
C02379=1076.444,367.613,399.687,175.754,30.239,155.352
C02380=1076.451,367.861,399.649,175.759,30.246,155.354
C02381=1076.457,368.107,399.612,175.762,30.252,155.355
C02382=1076.463,368.355,399.575,175.766,30.258,155.356
C02383=1076.470,368.602,399.537,175.769,30.264,155.357
C02384=1076.476,368.849,399.500,175.773,30.271,155.359
C02385=1076.482,369.096,399.463,175.777,30.277,155.360
C02386=1076.489,369.343,399.425,175.780,30.283,155.361
C02387=1076.495,369.590,399.389,175.785,30.289,155.362
C02388=1076.501,369.837,399.351,175.788,30.296,155.363
C02389=1076.508,370.084,399.313,175.791,30.302,155.365
C02390=1076.514,370.331,399.276,175.796,30.309,155.366
C02391=1076.521,370.579,399.239,175.799,30.315,155.367
C02392=1076.527,370.825,399.201,175.803,30.321,155.368
C02393=1076.533,371.048,399.168,175.806,30.327,155.369
C02394=1076.538,371.270,399.133,175.810,30.333,155.371
C02395=1076.545,371.493,399.100,175.813,30.338,155.372
C02396=1076.551,371.715,399.066,175.816,30.344,155.373
C02397=1076.556,371.937,399.032,175.820,30.350,155.374
C02398=1076.562,372.160,398.999,175.823,30.356,155.375
C02399=1076.568,372.383,398.964,175.827,30.362,155.376
C02400=1076.574,372.605,398.931,175.829,30.368,155.377
C02401=1076.580,372.852,398.893,175.834,30.374,155.379
C02402=1076.587,373.099,398.855,175.837,30.380,155.380
C02403=1076.594,373.346,398.817,175.842,30.387,155.381
C02404=1076.600,373.593,398.780,175.845,30.393,155.382
C02405=1076.607,373.840,398.742,175.848,30.400,155.384
C02406=1076.613,374.087,398.704,175.853,30.407,155.385
C02407=1076.619,374.334,398.666,175.856,30.413,155.386
C02408=1076.625,374.581,398.628,175.860,30.420,155.388
C02409=1076.632,374.828,398.590,175.864,30.427,155.389
C02410=1076.639,375.074,398.552,175.867,30.433,155.390
C02411=1076.645,375.322,398.514,175.871,30.440,155.392
C02412=1076.651,375.569,398.477,175.875,30.447,155.393
C02413=1076.657,375.816,398.438,175.879,30.453,155.394
C02414=1076.663,376.063,398.401,175.883,30.460,155.396
C02415=1076.670,376.310,398.362,175.886,30.467,155.397
C02416=1076.677,376.556,398.325,175.890,30.473,155.398
C02417=1076.683,376.804,398.287,175.894,30.480,155.400
C02418=1076.690,377.050,398.248,175.898,30.487,155.401
C02419=1076.696,377.297,398.210,175.902,30.494,155.402
C02420=1076.703,377.545,398.172,175.906,30.501,155.404
C02421=1076.709,377.791,398.133,175.910,30.507,155.405
C02422=1076.715,378.038,398.095,175.913,30.514,155.406
C02423=1076.722,378.285,398.056,175.917,30.521,155.408
C02424=1076.729,378.532,398.018,175.921,30.528,155.409
C02425=1076.736,378.778,397.980,175.925,30.535,155.410
C02426=1076.742,379.026,397.942,175.929,30.541,155.412
C02427=1076.749,379.272,397.903,175.932,30.548,155.413
C02428=1076.755,379.519,397.866,175.937,30.555,155.415
C02429=1076.762,379.766,397.827,175.940,30.562,155.416
C02430=1076.768,380.014,397.789,175.945,30.569,155.417
C02431=1076.775,380.260,397.750,175.948,30.576,155.419
C02432=1076.781,380.507,397.712,175.952,30.583,155.420
C02433=1076.788,380.754,397.673,175.956,30.590,155.421
C02434=1076.794,381.001,397.634,175.960,30.597,155.423
C02435=1076.801,381.248,397.596,175.964,30.604,155.424
C02436=1076.807,381.494,397.558,175.968,30.611,155.426
C02437=1076.814,381.741,397.519,175.972,30.618,155.427
C02438=1076.821,381.988,397.480,175.976,30.625,155.428
C02439=1076.827,382.235,397.442,175.979,30.632,155.430
C02440=1076.834,382.482,397.403,175.984,30.639,155.431
C02441=1076.840,382.729,397.364,175.987,30.646,155.433
C02442=1076.846,382.975,397.325,175.992,30.653,155.434
C02443=1076.853,383.222,397.287,175.995,30.660,155.436
C02444=1076.860,383.469,397.248,176.000,30.668,155.437
C02445=1076.867,383.716,397.209,176.003,30.675,155.439
C02446=1076.872,383.962,397.170,176.007,30.682,155.440
C02447=1076.879,384.209,397.131,176.011,30.690,155.442
C02448=1076.886,384.456,397.092,176.015,30.697,155.443
C02449=1076.892,384.693,397.054,176.019,30.704,155.444
C02450=1076.898,384.930,397.017,176.023,30.711,155.446
C02451=1076.905,385.167,396.980,176.027,30.718,155.447
C02452=1076.910,385.404,396.942,176.030,30.725,155.449
C02453=1076.918,385.641,396.905,176.034,30.732,155.450
C02454=1076.923,385.878,396.867,176.038,30.739,155.451
C02455=1076.930,386.115,396.830,176.042,30.746,155.453
C02456=1076.936,386.351,396.792,176.046,30.753,155.454
C02457=1076.943,386.598,396.753,176.049,30.760,155.456
C02458=1076.950,386.845,396.714,176.054,30.768,155.457
C02459=1076.956,387.092,396.675,176.058,30.775,155.459
C02460=1076.963,387.338,396.635,176.062,30.782,155.460
C02461=1076.970,387.585,396.596,176.066,30.790,155.462
C02462=1076.976,387.832,396.557,176.070,30.797,155.463
C02463=1076.983,388.078,396.517,176.074,30.805,155.465
C02464=1076.990,388.325,396.479,176.078,30.812,155.466
C02465=1076.996,388.572,396.439,176.082,30.820,155.468
C02466=1077.003,388.819,396.400,176.086,30.827,155.470
C02467=1077.010,389.065,396.361,176.091,30.835,155.471
C02468=1077.016,389.312,396.321,176.094,30.842,155.473
C02469=1077.023,389.559,396.282,176.098,30.850,155.474
C02470=1077.029,389.805,396.242,176.103,30.858,155.476
C02471=1077.037,390.053,396.202,176.106,30.865,155.477
C02472=1077.044,390.299,396.163,176.111,30.873,155.479
C02473=1077.050,390.546,396.123,176.115,30.880,155.480
C02474=1077.057,390.792,396.084,176.119,30.888,155.482
C02475=1077.063,391.039,396.044,176.123,30.896,155.484
C02476=1077.070,391.286,396.005,176.128,30.903,155.485
C02477=1077.077,391.532,395.965,176.131,30.911,155.487
C02478=1077.084,391.778,395.925,176.135,30.919,155.488
C02479=1077.090,392.026,395.885,176.140,30.927,155.490
C02480=1077.097,392.272,395.846,176.144,30.934,155.492
C02481=1077.104,392.519,395.806,176.148,30.942,155.493
C02482=1077.110,392.765,395.765,176.152,30.950,155.495
C02483=1077.117,393.012,395.726,176.157,30.958,155.496
C02484=1077.124,393.259,395.686,176.160,30.966,155.498
C02485=1077.130,393.506,395.646,176.165,30.974,155.500
C02486=1077.137,393.752,395.606,176.169,30.982,155.501
C02487=1077.144,393.999,395.566,176.174,30.989,155.503
C02488=1077.150,394.245,395.526,176.177,30.997,155.505
C02489=1077.158,394.492,395.486,176.181,31.005,155.506
C02490=1077.164,394.739,395.446,176.186,31.013,155.508
C02491=1077.171,394.985,395.406,176.190,31.022,155.510
C02492=1077.178,395.232,395.365,176.194,31.029,155.511
C02493=1077.185,395.479,395.326,176.198,31.037,155.513
C02494=1077.191,395.725,395.286,176.203,31.046,155.515
C02495=1077.197,395.972,395.246,176.207,31.054,155.516
C02496=1077.205,396.218,395.204,176.211,31.062,155.518
C02497=1077.211,396.465,395.164,176.215,31.070,155.520
C02498=1077.218,396.711,395.124,176.220,31.079,155.522
C02499=1077.225,396.958,395.084,176.224,31.087,155.523
C02500=1077.232,397.205,395.044,176.229,31.095,155.525
C02501=1077.239,397.451,395.003,176.232,31.103,155.527
C02502=1077.245,397.698,394.963,176.237,31.111,155.528
C02503=1077.252,397.944,394.922,176.241,31.120,155.530
C02504=1077.259,398.191,394.881,176.245,31.128,155.532
C02505=1077.266,398.436,394.841,176.250,31.136,155.534
C02506=1077.272,398.679,394.801,176.253,31.144,155.535
C02507=1077.279,398.924,394.761,176.258,31.153,155.537
C02508=1077.286,399.168,394.721,176.262,31.161,155.539
C02509=1077.293,399.412,394.681,176.267,31.169,155.541
C02510=1077.300,399.657,394.640,176.271,31.178,155.542
C02511=1077.307,399.901,394.600,176.275,31.186,155.544
C02512=1077.312,400.145,394.560,176.279,31.194,155.546
C02513=1077.320,400.392,394.518,176.284,31.203,155.548
C02514=1077.326,400.638,394.478,176.288,31.212,155.550
C02515=1077.333,400.885,394.437,176.293,31.220,155.551
C02516=1077.340,401.131,394.396,176.297,31.229,155.553
C02517=1077.347,401.378,394.356,176.302,31.237,155.555
C02518=1077.354,401.625,394.314,176.305,31.245,155.557
C02519=1077.361,401.871,394.274,176.310,31.254,155.559
C02520=1077.368,402.117,394.232,176.314,31.263,155.561
C02521=1077.375,402.364,394.192,176.319,31.271,155.562
C02522=1077.381,402.611,394.150,176.323,31.280,155.564
C02523=1077.388,402.857,394.109,176.328,31.289,155.566
C02524=1077.395,403.103,394.068,176.332,31.298,155.568
C02525=1077.402,403.350,394.027,176.337,31.306,155.570
C02526=1077.410,403.596,393.986,176.341,31.315,155.572
C02527=1077.416,403.843,393.946,176.346,31.324,155.574
C02528=1077.423,404.090,393.904,176.350,31.333,155.576
C02529=1077.430,404.336,393.863,176.355,31.342,155.577
C02530=1077.437,404.583,393.821,176.359,31.351,155.579
C02531=1077.444,404.829,393.781,176.364,31.360,155.581
C02532=1077.450,405.076,393.739,176.368,31.368,155.583
C02533=1077.458,405.322,393.697,176.373,31.377,155.585
C02534=1077.465,405.568,393.656,176.377,31.387,155.587
C02535=1077.471,405.815,393.614,176.382,31.396,155.589
C02536=1077.479,406.061,393.573,176.386,31.405,155.591
C02537=1077.485,406.308,393.531,176.391,31.414,155.593
C02538=1077.492,406.555,393.490,176.395,31.423,155.595
C02539=1077.499,406.800,393.448,176.400,31.432,155.597
C02540=1077.506,407.047,393.406,176.405,31.441,155.599
C02541=1077.513,407.293,393.365,176.409,31.450,155.601
C02542=1077.520,407.540,393.323,176.414,31.460,155.603
C02543=1077.527,407.786,393.281,176.418,31.469,155.605
C02544=1077.534,408.033,393.240,176.423,31.478,155.607
C02545=1077.541,408.278,393.198,176.427,31.488,155.609
C02546=1077.547,408.525,393.156,176.433,31.497,155.611
C02547=1077.554,408.772,393.114,176.437,31.506,155.613
C02548=1077.562,409.018,393.072,176.442,31.516,155.615
C02549=1077.568,409.265,393.030,176.446,31.525,155.617
C02550=1077.576,409.511,392.989,176.451,31.535,155.619
C02551=1077.583,409.757,392.946,176.455,31.544,155.621
C02552=1077.590,410.003,392.904,176.460,31.553,155.623
C02553=1077.597,410.250,392.862,176.465,31.563,155.625
C02554=1077.604,410.497,392.820,176.470,31.573,155.627
C02555=1077.611,410.743,392.778,176.475,31.582,155.629
C02556=1077.618,410.989,392.736,176.479,31.591,155.631
C02557=1077.625,411.236,392.693,176.484,31.601,155.634
C02558=1077.632,411.482,392.652,176.488,31.611,155.636
C02559=1077.639,411.728,392.609,176.494,31.620,155.638
C02560=1077.647,411.974,392.567,176.499,31.630,155.640
C02561=1077.653,412.220,392.525,176.503,31.640,155.642
C02562=1077.660,412.465,392.483,176.508,31.650,155.644
C02563=1077.667,412.711,392.441,176.513,31.659,155.646
C02564=1077.675,412.956,392.398,176.518,31.669,155.648
C02565=1077.682,413.202,392.357,176.522,31.679,155.650
C02566=1077.688,413.448,392.314,176.527,31.689,155.653
C02567=1077.696,413.693,392.272,176.533,31.699,155.655
C02568=1077.703,413.939,392.230,176.537,31.709,155.657
C02569=1077.710,414.185,392.187,176.542,31.718,155.659
C02570=1077.717,414.430,392.144,176.546,31.728,155.661
C02571=1077.724,414.677,392.101,176.552,31.738,155.663
C02572=1077.732,414.923,392.059,176.557,31.748,155.666
C02573=1077.739,415.170,392.017,176.561,31.758,155.668
C02574=1077.746,415.416,391.974,176.567,31.768,155.670
C02575=1077.753,415.662,391.931,176.571,31.778,155.672
C02576=1077.761,415.909,391.888,176.576,31.789,155.675
C02577=1077.768,416.155,391.845,176.582,31.799,155.677
C02578=1077.775,416.401,391.802,176.586,31.809,155.679
C02579=1077.782,416.647,391.760,176.592,31.819,155.681
C02580=1077.789,416.893,391.716,176.597,31.829,155.684
C02581=1077.796,417.140,391.673,176.601,31.840,155.686
C02582=1077.803,417.385,391.630,176.607,31.850,155.688
C02583=1077.810,417.632,391.588,176.612,31.860,155.691
C02584=1077.818,417.878,391.544,176.617,31.871,155.693
C02585=1077.825,418.124,391.501,176.622,31.881,155.695
C02586=1077.832,418.370,391.458,176.626,31.891,155.697
C02587=1077.840,418.616,391.415,176.632,31.902,155.700
C02588=1077.847,418.862,391.372,176.637,31.913,155.702
C02589=1077.854,419.109,391.328,176.642,31.923,155.705
C02590=1077.862,419.355,391.285,176.647,31.934,155.707
C02591=1077.868,419.601,391.243,176.653,31.945,155.709
C02592=1077.876,419.847,391.199,176.657,31.955,155.712
C02593=1077.883,420.093,391.156,176.663,31.966,155.714
C02594=1077.891,420.339,391.112,176.668,31.976,155.716
C02595=1077.898,420.585,391.069,176.673,31.987,155.719
C02596=1077.906,420.831,391.025,176.678,31.998,155.721
C02597=1077.912,421.077,390.981,176.684,32.009,155.724
C02598=1077.920,421.324,390.938,176.689,32.020,155.726
C02599=1077.927,421.569,390.894,176.694,32.031,155.729
C02600=1077.935,421.816,390.851,176.700,32.042,155.731
C02601=1077.942,422.061,390.808,176.705,32.052,155.733
C02602=1077.949,422.308,390.763,176.710,32.063,155.736
C02603=1077.957,422.554,390.720,176.715,32.074,155.738
C02604=1077.964,422.800,390.676,176.721,32.086,155.741
C02605=1077.971,423.045,390.632,176.726,32.097,155.743
C02606=1077.979,423.292,390.588,176.731,32.107,155.746
C02607=1077.987,423.538,390.545,176.737,32.119,155.748
C02608=1077.993,423.783,390.500,176.743,32.130,155.751
C02609=1078.001,424.030,390.457,176.747,32.141,155.754
C02610=1078.007,424.276,390.413,176.753,32.153,155.756
C02611=1078.016,424.521,390.368,176.759,32.164,155.759
C02612=1078.023,424.768,390.325,176.764,32.175,155.761
C02613=1078.030,425.013,390.280,176.769,32.186,155.764
C02614=1078.038,425.260,390.237,176.775,32.198,155.766
C02615=1078.045,425.506,390.192,176.780,32.209,155.769
C02616=1078.053,425.751,390.147,176.786,32.221,155.772
C02617=1078.061,426.013,390.101,176.791,32.233,155.774
C02618=1078.069,426.276,390.053,176.797,32.245,155.777
C02619=1078.077,426.538,390.006,176.804,32.258,155.780
C02620=1078.085,426.799,389.959,176.810,32.270,155.783
C02621=1078.092,427.046,389.915,176.815,32.282,155.785
C02622=1078.100,427.292,389.870,176.820,32.293,155.788
C02623=1078.108,427.538,389.826,176.826,32.305,155.791
C02624=1078.115,427.784,389.781,176.832,32.317,155.793
C02625=1078.123,428.029,389.737,176.838,32.329,155.796
C02626=1078.130,428.275,389.692,176.843,32.341,155.799
C02627=1078.138,428.521,389.647,176.848,32.352,155.802
C02628=1078.145,428.767,389.603,176.854,32.364,155.804
C02629=1078.153,429.013,389.558,176.860,32.376,155.807
C02630=1078.161,429.258,389.513,176.866,32.388,155.810
C02631=1078.168,429.504,389.468,176.872,32.400,155.813
C02632=1078.175,429.750,389.423,176.877,32.412,155.815
C02633=1078.182,429.996,389.379,176.883,32.424,155.818
C02634=1078.190,430.241,389.334,176.889,32.437,155.821
C02635=1078.198,430.487,389.289,176.895,32.449,155.824
C02636=1078.205,430.733,389.244,176.900,32.461,155.827
C02637=1078.213,430.978,389.199,176.906,32.473,155.829
C02638=1078.221,431.224,389.154,176.912,32.486,155.832
C02639=1078.228,431.470,389.109,176.917,32.498,155.835
C02640=1078.236,431.716,389.063,176.923,32.510,155.838
C02641=1078.244,431.962,389.019,176.929,32.523,155.841
C02642=1078.252,432.208,388.973,176.935,32.535,155.844
C02643=1078.259,432.454,388.928,176.941,32.548,155.847
C02644=1078.267,432.699,388.882,176.947,32.560,155.849
C02645=1078.275,432.945,388.837,176.953,32.573,155.852
C02646=1078.282,433.191,388.792,176.959,32.586,155.855
C02647=1078.290,433.436,388.746,176.965,32.598,155.858
C02648=1078.297,433.681,388.701,176.971,32.611,155.861
C02649=1078.305,433.927,388.655,176.978,32.624,155.864
C02650=1078.313,434.172,388.609,176.984,32.637,155.867
C02651=1078.321,434.419,388.564,176.989,32.649,155.870
C02652=1078.328,434.665,388.518,176.995,32.663,155.873
C02653=1078.336,434.910,388.473,177.001,32.675,155.876
C02654=1078.343,435.155,388.427,177.007,32.688,155.879
C02655=1078.351,435.401,388.381,177.013,32.701,155.882
C02656=1078.359,435.647,388.335,177.019,32.714,155.885
C02657=1078.367,435.892,388.290,177.025,32.727,155.889
C02658=1078.375,436.137,388.243,177.032,32.741,155.892
C02659=1078.383,436.383,388.198,177.038,32.754,155.895
C02660=1078.391,436.629,388.152,177.044,32.767,155.898
C02661=1078.398,436.874,388.106,177.050,32.780,155.901
C02662=1078.406,437.120,388.060,177.056,32.794,155.904
C02663=1078.414,437.365,388.013,177.063,32.807,155.907
C02664=1078.422,437.611,387.967,177.070,32.820,155.910
C02665=1078.430,437.857,387.921,177.076,32.834,155.913
C02666=1078.438,438.102,387.875,177.083,32.847,155.917
C02667=1078.445,438.347,387.829,177.089,32.861,155.920
C02668=1078.454,438.593,387.783,177.095,32.874,155.923
C02669=1078.462,438.838,387.737,177.101,32.888,155.926
C02670=1078.470,439.084,387.690,177.108,32.902,155.930
C02671=1078.478,439.330,387.643,177.114,32.915,155.933
C02672=1078.486,439.575,387.597,177.120,32.929,155.936
C02673=1078.497,439.941,387.528,177.130,32.950,155.941
C02674=1078.510,440.308,387.458,177.140,32.970,155.946
C02675=1078.521,440.674,387.388,177.150,32.992,155.951
C02676=1078.533,441.039,387.319,177.160,33.013,155.956
C02677=1078.542,441.285,387.272,177.166,33.027,155.959
C02678=1078.549,441.531,387.225,177.172,33.041,155.963
C02679=1078.557,441.776,387.178,177.180,33.055,155.966
C02680=1078.565,442.021,387.131,177.186,33.069,155.969
C02681=1078.574,442.267,387.084,177.193,33.084,155.973
C02682=1078.581,442.512,387.037,177.199,33.098,155.976
C02683=1078.589,442.758,386.991,177.206,33.113,155.980
C02684=1078.597,443.003,386.943,177.213,33.127,155.983
C02685=1078.606,443.248,386.896,177.220,33.141,155.987
C02686=1078.613,443.493,386.849,177.226,33.156,155.990
C02687=1078.622,443.739,386.802,177.233,33.171,155.994
C02688=1078.630,443.984,386.754,177.241,33.185,155.997
C02689=1078.639,444.230,386.707,177.247,33.200,156.001
C02690=1078.646,444.474,386.660,177.254,33.215,156.004
C02691=1078.655,444.720,386.613,177.261,33.230,156.008
C02692=1078.663,444.965,386.565,177.268,33.244,156.011
C02693=1078.670,445.211,386.518,177.275,33.260,156.015
C02694=1078.679,445.456,386.470,177.282,33.275,156.019
C02695=1078.687,445.701,386.422,177.289,33.290,156.022
C02696=1078.696,445.946,386.374,177.296,33.305,156.026
C02697=1078.704,446.191,386.327,177.303,33.320,156.030
C02698=1078.712,446.436,386.280,177.310,33.335,156.033
C02699=1078.720,446.681,386.232,177.316,33.350,156.037
C02700=1078.728,446.926,386.184,177.323,33.365,156.041
C02701=1078.737,447.171,386.136,177.328,33.381,156.045
C02702=1078.745,447.416,386.088,177.335,33.396,156.048
C02703=1078.754,447.662,386.040,177.340,33.411,156.052
C02704=1078.762,447.908,385.992,177.346,33.426,156.056
C02705=1078.771,448.152,385.944,177.350,33.441,156.059
C02706=1078.779,448.398,385.896,177.355,33.456,156.063
C02707=1078.787,448.643,385.848,177.360,33.471,156.067
C02708=1078.795,448.887,385.799,177.364,33.486,156.071
C02709=1078.805,449.132,385.752,177.368,33.501,156.074
C02710=1078.815,449.377,385.705,177.373,33.515,156.078
C02711=1078.827,449.623,385.659,177.376,33.528,156.081
C02712=1078.841,449.869,385.614,177.381,33.541,156.085
C02713=1078.478,449.864,385.387,177.357,33.704,156.128
C02714=1078.459,449.535,385.447,177.351,33.687,156.123
C02715=1078.444,449.207,385.509,177.345,33.669,156.119
C02716=1078.431,448.882,385.573,177.340,33.649,156.114
C02717=1078.420,448.556,385.637,177.334,33.629,156.109
C02718=1078.412,448.311,385.685,177.329,33.614,156.105
C02719=1078.403,448.066,385.732,177.324,33.599,156.102
C02720=1078.395,447.821,385.780,177.318,33.584,156.098
C02721=1078.387,447.575,385.828,177.313,33.569,156.094
C02722=1078.379,447.330,385.876,177.307,33.554,156.090
C02723=1078.371,447.086,385.925,177.302,33.539,156.087
C02724=1078.362,446.841,385.973,177.295,33.523,156.083
C02725=1078.354,446.595,386.021,177.288,33.508,156.079
C02726=1078.346,446.350,386.068,177.282,33.493,156.075
C02727=1078.337,446.105,386.115,177.275,33.478,156.072
C02728=1078.329,445.860,386.164,177.267,33.463,156.068
C02729=1078.321,445.614,386.212,177.261,33.448,156.064
C02730=1078.313,445.369,386.260,177.253,33.433,156.061
C02731=1078.304,445.124,386.307,177.246,33.418,156.057
C02732=1078.296,444.878,386.354,177.239,33.403,156.053
C02733=1078.288,444.633,386.402,177.232,33.388,156.050
C02734=1078.279,444.388,386.450,177.224,33.373,156.046
C02735=1078.271,444.143,386.497,177.218,33.359,156.043
C02736=1078.263,443.898,386.544,177.211,33.343,156.039
C02737=1078.255,443.653,386.592,177.204,33.329,156.036
C02738=1078.246,443.408,386.639,177.197,33.315,156.032
C02739=1078.239,443.162,386.686,177.190,33.300,156.029
C02740=1078.230,442.916,386.733,177.183,33.285,156.025
C02741=1078.222,442.672,386.781,177.176,33.271,156.022
C02742=1078.214,442.426,386.827,177.170,33.256,156.018
C02743=1078.206,442.180,386.875,177.162,33.242,156.015
C02744=1078.198,441.936,386.921,177.156,33.228,156.011
C02745=1078.190,441.690,386.968,177.150,33.213,156.008
C02746=1078.181,441.445,387.016,177.142,33.199,156.004
C02747=1078.173,441.199,387.063,177.136,33.185,156.001
C02748=1078.166,440.954,387.110,177.129,33.171,155.998
C02749=1078.157,440.709,387.156,177.123,33.157,155.994
C02750=1078.149,440.441,387.207,177.115,33.142,155.991
C02751=1078.140,440.173,387.258,177.108,33.127,155.987
C02752=1078.131,439.906,387.309,177.101,33.111,155.983
C02753=1078.123,439.637,387.360,177.094,33.096,155.980
C02754=1078.115,439.392,387.406,177.087,33.082,155.977
C02755=1078.107,439.146,387.452,177.080,33.069,155.973
C02756=1078.099,438.901,387.499,177.074,33.055,155.970
C02757=1078.091,438.656,387.546,177.068,33.041,155.967
C02758=1078.083,438.410,387.592,177.061,33.028,155.964
C02759=1078.075,438.165,387.638,177.055,33.014,155.960
C02760=1078.066,437.919,387.684,177.048,33.001,155.957
C02761=1078.058,437.674,387.731,177.042,32.987,155.954
C02762=1078.051,437.428,387.777,177.035,32.974,155.951
C02763=1078.042,437.183,387.823,177.029,32.961,155.948
C02764=1078.035,436.937,387.869,177.023,32.947,155.944
C02765=1078.027,436.691,387.915,177.017,32.934,155.941
C02766=1078.019,436.446,387.962,177.010,32.920,155.938
C02767=1078.011,436.201,388.008,177.004,32.908,155.935
C02768=1078.003,435.955,388.054,176.997,32.894,155.932
C02769=1077.996,435.709,388.099,176.991,32.881,155.929
C02770=1077.988,435.464,388.145,176.985,32.868,155.926
C02771=1077.980,435.218,388.191,176.979,32.855,155.923
C02772=1077.972,434.972,388.236,176.972,32.842,155.920
C02773=1077.964,434.727,388.282,176.966,32.829,155.917
C02774=1077.957,434.481,388.328,176.960,32.816,155.914
C02775=1077.949,434.236,388.373,176.954,32.803,155.911
C02776=1077.941,433.990,388.419,176.948,32.791,155.908
C02777=1077.933,433.744,388.465,176.942,32.778,155.905
C02778=1077.926,433.499,388.511,176.936,32.765,155.902
C02779=1077.918,433.253,388.556,176.930,32.752,155.899
C02780=1077.910,433.008,388.602,176.924,32.740,155.896
C02781=1077.903,432.762,388.647,176.918,32.727,155.893
C02782=1077.895,432.517,388.693,176.912,32.714,155.890
C02783=1077.888,432.271,388.738,176.906,32.702,155.887
C02784=1077.880,432.024,388.784,176.900,32.689,155.884
C02785=1077.871,431.779,388.829,176.894,32.677,155.881
C02786=1077.864,431.533,388.874,176.888,32.665,155.878
C02787=1077.857,431.288,388.919,176.882,32.652,155.876
C02788=1077.849,431.042,388.964,176.876,32.640,155.873
C02789=1077.841,430.797,389.009,176.870,32.628,155.870
C02790=1077.833,430.550,389.054,176.864,32.615,155.867
C02791=1077.826,430.304,389.099,176.858,32.603,155.864
C02792=1077.819,430.059,389.145,176.852,32.591,155.861
C02793=1077.810,429.813,389.189,176.846,32.579,155.859
C02794=1077.803,429.567,389.234,176.840,32.567,155.856
C02795=1077.796,429.321,389.279,176.835,32.555,155.853
C02796=1077.787,429.076,389.324,176.830,32.543,155.850
C02797=1077.780,428.830,389.369,176.824,32.530,155.847
C02798=1077.773,428.584,389.414,176.818,32.519,155.845
C02799=1077.765,428.339,389.458,176.812,32.507,155.842
C02800=1077.758,428.093,389.503,176.806,32.495,155.839
C02801=1077.751,427.847,389.548,176.801,32.483,155.837
C02802=1077.743,427.601,389.592,176.795,32.471,155.834
C02803=1077.735,427.355,389.637,176.789,32.460,155.831
C02804=1077.727,427.109,389.681,176.783,32.448,155.829
C02805=1077.720,426.863,389.726,176.778,32.437,155.826
C02806=1077.711,426.600,389.773,176.772,32.424,155.823
C02807=1077.704,426.336,389.821,176.766,32.412,155.820
C02808=1077.696,426.073,389.868,176.760,32.399,155.817
C02809=1077.688,425.809,389.916,176.754,32.387,155.815
C02810=1077.680,425.563,389.960,176.748,32.376,155.812
C02811=1077.673,425.317,390.004,176.743,32.364,155.809
C02812=1077.665,425.071,390.049,176.738,32.353,155.807
C02813=1077.657,424.825,390.092,176.732,32.341,155.804
C02814=1077.650,424.579,390.137,176.726,32.330,155.802
C02815=1077.642,424.333,390.180,176.720,32.319,155.799
C02816=1077.636,424.087,390.225,176.716,32.307,155.796
C02817=1077.628,423.841,390.269,176.710,32.296,155.794
C02818=1077.620,423.595,390.313,176.705,32.285,155.791
C02819=1077.613,423.349,390.357,176.699,32.274,155.789
C02820=1077.606,423.103,390.400,176.693,32.263,155.786
C02821=1077.598,422.858,390.444,176.689,32.251,155.784
C02822=1077.591,422.611,390.489,176.683,32.240,155.781
C02823=1077.583,422.365,390.532,176.677,32.229,155.779
C02824=1077.576,422.119,390.576,176.672,32.218,155.776
C02825=1077.569,421.873,390.620,176.666,32.207,155.774
C02826=1077.562,421.627,390.664,176.662,32.196,155.771
C02827=1077.554,421.381,390.707,176.656,32.185,155.769
C02828=1077.547,421.135,390.751,176.651,32.175,155.766
C02829=1077.540,420.889,390.795,176.645,32.164,155.764
C02830=1077.533,420.643,390.838,176.641,32.153,155.762
C02831=1077.525,420.397,390.882,176.635,32.142,155.759
C02832=1077.518,420.151,390.925,176.629,32.132,155.757
C02833=1077.510,419.905,390.969,176.624,32.121,155.754
C02834=1077.503,419.659,391.012,176.619,32.110,155.752
C02835=1077.495,419.412,391.055,176.614,32.100,155.750
C02836=1077.488,419.166,391.098,176.609,32.089,155.747
C02837=1077.480,418.920,391.142,176.603,32.079,155.745
C02838=1077.473,418.674,391.185,176.599,32.068,155.743
C02839=1077.466,418.427,391.228,176.593,32.057,155.740
C02840=1077.459,418.182,391.271,176.588,32.047,155.738
C02841=1077.451,417.936,391.314,176.583,32.037,155.736
C02842=1077.444,417.689,391.357,176.578,32.026,155.733
C02843=1077.437,417.443,391.400,176.572,32.016,155.731
C02844=1077.430,417.198,391.444,176.568,32.005,155.729
C02845=1077.422,416.951,391.487,176.563,31.995,155.726
C02846=1077.415,416.705,391.530,176.557,31.985,155.724
C02847=1077.408,416.459,391.572,176.552,31.975,155.722
C02848=1077.401,416.213,391.616,176.548,31.965,155.720
C02849=1077.394,415.966,391.659,176.542,31.954,155.717
C02850=1077.387,415.720,391.701,176.537,31.944,155.715
C02851=1077.380,415.474,391.744,176.533,31.934,155.713
C02852=1077.373,415.228,391.787,176.527,31.924,155.711
C02853=1077.365,414.981,391.830,176.522,31.914,155.708
C02854=1077.358,414.735,391.873,176.518,31.903,155.706
C02855=1077.350,414.489,391.915,176.512,31.893,155.704
C02856=1077.344,414.243,391.958,176.507,31.884,155.702
C02857=1077.336,413.996,392.000,176.503,31.874,155.699
C02858=1077.329,413.750,392.043,176.497,31.864,155.697
C02859=1077.322,413.504,392.085,176.492,31.854,155.695
C02860=1077.315,413.257,392.127,176.488,31.844,155.693
C02861=1077.308,413.012,392.171,176.483,31.834,155.691
C02862=1077.300,412.766,392.213,176.477,31.825,155.689
C02863=1077.293,412.520,392.255,176.473,31.815,155.687
C02864=1077.285,412.273,392.297,176.468,31.805,155.684
C02865=1077.279,412.026,392.339,176.464,31.796,155.682
C02866=1077.272,411.780,392.382,176.458,31.785,155.680
C02867=1077.264,411.534,392.424,176.453,31.776,155.678
C02868=1077.257,411.287,392.466,176.449,31.767,155.676
C02869=1077.250,411.041,392.509,176.444,31.757,155.674
C02870=1077.243,410.795,392.551,176.439,31.747,155.672
C02871=1077.236,410.548,392.593,176.434,31.738,155.670
C02872=1077.229,410.302,392.635,176.429,31.728,155.668
C02873=1077.222,410.056,392.677,176.425,31.719,155.665
C02874=1077.215,409.810,392.720,176.420,31.709,155.663
C02875=1077.208,409.563,392.761,176.415,31.700,155.661
C02876=1077.201,409.317,392.803,176.411,31.691,155.659
C02877=1077.194,409.070,392.845,176.406,31.681,155.657
C02878=1077.187,408.824,392.887,176.400,31.671,155.655
C02879=1077.180,408.577,392.929,176.396,31.662,155.653
C02880=1077.173,408.332,392.971,176.391,31.653,155.651
C02881=1077.167,408.085,393.012,176.387,31.643,155.649
C02882=1077.159,407.839,393.054,176.382,31.634,155.647
C02883=1077.152,407.592,393.096,176.377,31.625,155.645
C02884=1077.145,407.346,393.138,176.373,31.616,155.643
C02885=1077.138,407.099,393.180,176.368,31.606,155.641
C02886=1077.131,406.853,393.221,176.364,31.597,155.639
C02887=1077.125,406.607,393.263,176.359,31.588,155.637
C02888=1077.117,406.360,393.305,176.355,31.579,155.635
C02889=1077.111,406.113,393.346,176.350,31.570,155.633
C02890=1077.104,405.867,393.388,176.345,31.561,155.631
C02891=1077.096,405.621,393.430,176.341,31.552,155.629
C02892=1077.090,405.375,393.471,176.336,31.542,155.627
C02893=1077.083,405.128,393.512,176.332,31.534,155.625
C02894=1077.075,404.881,393.554,176.327,31.525,155.623
C02895=1077.069,404.635,393.595,176.323,31.516,155.621
C02896=1077.062,404.389,393.636,176.318,31.507,155.620
C02897=1077.055,404.142,393.677,176.313,31.498,155.618
C02898=1077.048,403.895,393.719,176.309,31.489,155.616
C02899=1077.041,403.649,393.760,176.304,31.480,155.614
C02900=1077.034,403.403,393.801,176.300,31.472,155.612
C02901=1077.027,403.156,393.843,176.295,31.463,155.610
C02902=1077.020,402.910,393.884,176.291,31.454,155.608
C02903=1077.013,402.664,393.925,176.286,31.445,155.606
C02904=1077.007,402.417,393.966,176.281,31.437,155.605
C02905=1076.999,402.170,394.008,176.277,31.428,155.603
C02906=1076.993,401.924,394.048,176.272,31.419,155.601
C02907=1076.986,401.677,394.089,176.269,31.411,155.599
C02908=1076.978,401.430,394.130,176.264,31.402,155.597
C02909=1076.972,401.185,394.171,176.260,31.393,155.595
C02910=1076.965,400.937,394.212,176.255,31.385,155.593
C02911=1076.958,400.691,394.253,176.251,31.376,155.592
C02912=1076.951,400.445,394.294,176.246,31.368,155.590
C02913=1076.945,400.198,394.335,176.242,31.359,155.588
C02914=1076.937,399.953,394.376,176.237,31.351,155.586
C02915=1076.930,399.708,394.415,176.233,31.342,155.584
C02916=1076.924,399.463,394.456,176.229,31.334,155.583
C02917=1076.917,399.219,394.497,176.224,31.325,155.581
C02918=1076.911,398.973,394.537,176.220,31.317,155.579
C02919=1076.904,398.728,394.577,176.215,31.309,155.577
C02920=1076.897,398.483,394.617,176.212,31.301,155.576
C02921=1076.891,398.239,394.658,176.207,31.293,155.574
C02922=1076.883,397.992,394.698,176.203,31.284,155.572
C02923=1076.876,397.745,394.738,176.198,31.275,155.570
C02924=1076.869,397.499,394.780,176.194,31.267,155.569
C02925=1076.863,397.252,394.820,176.190,31.259,155.567
C02926=1076.856,397.005,394.860,176.186,31.251,155.565
C02927=1076.849,396.758,394.901,176.181,31.243,155.563
C02928=1076.843,396.512,394.941,176.177,31.234,155.562
C02929=1076.836,396.265,394.982,176.173,31.227,155.560
C02930=1076.829,396.019,395.021,176.169,31.219,155.558
C02931=1076.822,395.773,395.062,176.164,31.210,155.557
C02932=1076.815,395.525,395.102,176.160,31.202,155.555
C02933=1076.809,395.279,395.143,176.156,31.194,155.553
C02934=1076.802,395.033,395.183,176.152,31.186,155.551
C02935=1076.794,394.786,395.223,176.147,31.178,155.550
C02936=1076.788,394.539,395.263,176.143,31.170,155.548
C02937=1076.782,394.293,395.303,176.139,31.162,155.546
C02938=1076.775,394.046,395.343,176.135,31.154,155.545
C02939=1076.768,393.800,395.383,176.130,31.146,155.543
C02940=1076.761,393.553,395.424,176.126,31.138,155.541
C02941=1076.755,393.307,395.464,176.122,31.130,155.540
C02942=1076.748,393.060,395.503,176.118,31.122,155.538
C02943=1076.741,392.812,395.543,176.113,31.114,155.537
C02944=1076.735,392.566,395.583,176.110,31.107,155.535
C02945=1076.728,392.320,395.623,176.105,31.098,155.533
C02946=1076.721,392.073,395.663,176.101,31.091,155.532
C02947=1076.714,391.827,395.702,176.097,31.083,155.530
C02948=1076.707,391.579,395.742,176.093,31.075,155.528
C02949=1076.701,391.333,395.782,176.088,31.067,155.527
C02950=1076.694,391.087,395.822,176.085,31.060,155.525
C02951=1076.688,390.839,395.861,176.080,31.052,155.524
C02952=1076.681,390.593,395.901,176.076,31.044,155.522
C02953=1076.674,390.347,395.940,176.072,31.037,155.520
C02954=1076.667,390.099,395.980,176.068,31.029,155.519
C02955=1076.660,389.853,396.020,176.063,31.022,155.517
C02956=1076.654,389.606,396.059,176.060,31.014,155.516
C02957=1076.647,389.360,396.099,176.055,31.006,155.514
C02958=1076.639,389.113,396.138,176.051,30.999,155.513
C02959=1076.633,388.866,396.178,176.047,30.991,155.511
C02960=1076.627,388.619,396.217,176.043,30.984,155.510
C02961=1076.619,388.373,396.256,176.038,30.976,155.508
C02962=1076.613,388.126,396.296,176.035,30.969,155.506
C02963=1076.606,387.880,396.335,176.030,30.961,155.505
C02964=1076.599,387.633,396.374,176.027,30.954,155.503
C02965=1076.593,387.386,396.413,176.022,30.947,155.502
C02966=1076.586,387.140,396.453,176.018,30.939,155.500
C02967=1076.579,386.893,396.492,176.014,30.932,155.499
C02968=1076.573,386.646,396.531,176.010,30.924,155.497
C02969=1076.566,386.400,396.571,176.006,30.917,155.496
C02970=1076.560,386.161,396.608,176.002,30.910,155.494
C02971=1076.554,385.923,396.646,175.998,30.903,155.493
C02972=1076.547,385.686,396.684,175.994,30.896,155.492
C02973=1076.541,385.449,396.721,175.990,30.889,155.490
C02974=1076.535,385.211,396.759,175.987,30.882,155.489
C02975=1076.528,384.973,396.796,175.982,30.875,155.487
C02976=1076.522,384.736,396.834,175.979,30.868,155.486
C02977=1076.516,384.498,396.872,175.975,30.860,155.484
C02978=1076.509,384.251,396.911,175.971,30.853,155.483
C02979=1076.503,384.005,396.949,175.967,30.846,155.481
C02980=1076.496,383.759,396.988,175.963,30.839,155.480
C02981=1076.490,383.511,397.028,175.959,30.832,155.479
C02982=1076.483,383.265,397.066,175.955,30.824,155.477
C02983=1076.476,383.018,397.105,175.951,30.817,155.476
C02984=1076.469,382.771,397.144,175.947,30.810,155.474
C02985=1076.464,382.525,397.183,175.943,30.803,155.473
C02986=1076.457,382.278,397.222,175.939,30.796,155.471
C02987=1076.450,382.031,397.261,175.935,30.788,155.470
C02988=1076.444,381.783,397.299,175.931,30.782,155.468
C02989=1076.437,381.537,397.337,175.927,30.774,155.467
C02990=1076.431,381.290,397.376,175.923,30.767,155.466
C02991=1076.424,381.044,397.415,175.919,30.760,155.464
C02992=1076.417,380.796,397.453,175.916,30.753,155.463
C02993=1076.410,380.549,397.492,175.911,30.746,155.461
C02994=1076.404,380.303,397.531,175.908,30.740,155.460
C02995=1076.398,380.056,397.569,175.904,30.733,155.459
C02996=1076.391,379.809,397.607,175.900,30.726,155.457
C02997=1076.384,379.562,397.646,175.896,30.719,155.456
C02998=1076.378,379.315,397.684,175.892,30.712,155.454
C02999=1076.371,379.069,397.723,175.888,30.705,155.453
C03000=1076.365,378.821,397.761,175.884,30.698,155.452
C03001=1076.357,378.575,397.799,175.880,30.691,155.450
C03002=1076.351,378.328,397.837,175.876,30.685,155.449
C03003=1076.345,378.081,397.876,175.873,30.678,155.447
C03004=1076.338,377.834,397.914,175.869,30.671,155.446
C03005=1076.332,377.588,397.952,175.865,30.664,155.445
C03006=1076.325,377.340,397.991,175.861,30.658,155.443
C03007=1076.319,377.093,398.029,175.857,30.650,155.442
C03008=1076.313,376.846,398.067,175.853,30.644,155.441
C03009=1076.306,376.599,398.105,175.850,30.637,155.439
C03010=1076.300,376.352,398.143,175.845,30.630,155.438
C03011=1076.293,376.106,398.181,175.842,30.623,155.437
C03012=1076.286,375.858,398.219,175.837,30.617,155.435
C03013=1076.280,375.612,398.257,175.834,30.610,155.434
C03014=1076.274,375.364,398.295,175.831,30.603,155.433
C03015=1076.268,375.118,398.334,175.826,30.597,155.431
C03016=1076.261,374.871,398.372,175.823,30.590,155.430
C03017=1076.254,374.624,398.409,175.819,30.584,155.429
C03018=1076.248,374.377,398.447,175.815,30.577,155.427
C03019=1076.241,374.129,398.485,175.811,30.570,155.426
C03020=1076.236,373.883,398.523,175.807,30.564,155.425
C03021=1076.229,373.635,398.561,175.803,30.557,155.424
C03022=1076.222,373.389,398.598,175.800,30.551,155.422
C03023=1076.216,373.141,398.636,175.796,30.544,155.421
C03024=1076.210,372.894,398.674,175.792,30.538,155.420
C03025=1076.203,372.647,398.712,175.789,30.531,155.418
C03026=1076.197,372.424,398.746,175.785,30.525,155.417
C03027=1076.191,372.202,398.780,175.782,30.519,155.416
C03028=1076.185,371.979,398.814,175.778,30.514,155.415
C03029=1076.179,371.755,398.848,175.775,30.508,155.414
C03030=1076.174,371.532,398.882,175.771,30.502,155.413
C03031=1076.168,371.309,398.916,175.768,30.496,155.412
C03032=1076.162,371.086,398.949,175.764,30.490,155.410
C03033=1076.156,370.862,398.984,175.762,30.485,155.409
C03034=1076.150,370.616,399.021,175.757,30.478,155.408
C03035=1076.143,370.369,399.059,175.754,30.472,155.407
C03036=1076.137,370.122,399.096,175.750,30.466,155.406
C03037=1076.131,369.875,399.133,175.746,30.459,155.404
C03038=1076.124,369.628,399.171,175.742,30.453,155.403
C03039=1076.118,369.381,399.209,175.739,30.446,155.402
C03040=1076.111,369.133,399.245,175.735,30.440,155.401
C03041=1076.105,368.886,399.283,175.731,30.434,155.399
C03042=1076.098,368.640,399.320,175.728,30.428,155.398
C03043=1076.092,368.392,399.358,175.724,30.421,155.397
C03044=1076.085,368.146,399.395,175.720,30.415,155.396
C03045=1076.079,367.897,399.432,175.716,30.409,155.395
C03046=1076.073,367.651,399.469,175.713,30.403,155.393
C03047=1076.067,367.404,399.506,175.710,30.396,155.392
C03048=1076.060,367.156,399.544,175.705,30.390,155.391
C03049=1076.053,366.909,399.580,175.702,30.383,155.390
C03050=1076.047,366.663,399.618,175.698,30.377,155.388
C03051=1076.041,366.416,399.655,175.695,30.371,155.387
C03052=1076.035,366.168,399.693,175.690,30.365,155.386
C03053=1076.028,365.921,399.729,175.687,30.359,155.385
C03054=1076.023,365.674,399.766,175.684,30.353,155.384
C03055=1076.016,365.427,399.803,175.680,30.347,155.383
C03056=1076.009,365.180,399.840,175.677,30.340,155.381
C03057=1076.003,364.932,399.877,175.672,30.334,155.380
C03058=1075.997,364.686,399.914,175.669,30.328,155.379
C03059=1075.991,364.439,399.951,175.665,30.322,155.378
C03060=1075.984,364.191,399.988,175.662,30.316,155.377
C03061=1075.978,363.944,400.025,175.658,30.310,155.375
C03062=1075.971,363.697,400.062,175.654,30.304,155.374
C03063=1075.965,363.450,400.098,175.651,30.298,155.373
C03064=1075.958,363.202,400.135,175.647,30.292,155.372
C03065=1075.952,362.955,400.172,175.644,30.286,155.371
C03066=1075.946,362.708,400.209,175.640,30.280,155.370
C03067=1075.940,362.461,400.245,175.636,30.274,155.369
C03068=1075.933,362.213,400.282,175.632,30.268,155.367
C03069=1075.927,361.966,400.318,175.629,30.262,155.366
C03070=1075.920,361.719,400.355,175.626,30.256,155.365
C03071=1075.914,361.472,400.391,175.622,30.250,155.364
C03072=1075.908,361.225,400.428,175.618,30.244,155.363
C03073=1075.902,360.978,400.465,175.614,30.239,155.362
C03074=1075.895,360.730,400.501,175.611,30.233,155.361
C03075=1075.889,360.483,400.538,175.607,30.227,155.359
C03076=1075.882,360.236,400.574,175.604,30.221,155.358
C03077=1075.876,359.989,400.611,175.601,30.215,155.357
C03078=1075.870,359.742,400.647,175.597,30.209,155.356
C03079=1075.863,359.495,400.684,175.593,30.203,155.355
C03080=1075.857,359.247,400.720,175.589,30.197,155.354
C03081=1075.851,359.000,400.756,175.586,30.191,155.353
C03082=1075.845,358.785,400.788,175.583,30.187,155.352
C03083=1075.840,358.570,400.819,175.580,30.182,155.351
C03084=1075.834,358.355,400.851,175.576,30.177,155.350
C03085=1075.829,358.141,400.882,175.574,30.171,155.349
C03086=1075.823,357.926,400.914,175.570,30.166,155.348
C03087=1075.817,357.711,400.945,175.568,30.161,155.347
C03088=1075.812,357.495,400.977,175.564,30.157,155.346
C03089=1075.807,357.282,401.008,175.561,30.152,155.345
C03090=1075.800,357.033,401.044,175.557,30.145,155.344
C03091=1075.794,356.786,401.081,175.554,30.140,155.343
C03092=1075.787,356.539,401.117,175.550,30.134,155.342
C03093=1075.781,356.291,401.153,175.547,30.128,155.341
C03094=1075.775,356.044,401.189,175.544,30.123,155.340
C03095=1075.769,355.797,401.225,175.540,30.117,155.339
C03096=1075.763,355.550,401.262,175.537,30.111,155.338
C03097=1075.757,355.302,401.297,175.533,30.106,155.337
C03098=1075.750,355.055,401.334,175.530,30.100,155.336
C03099=1075.744,354.808,401.369,175.526,30.095,155.335
C03100=1075.738,354.561,401.405,175.522,30.089,155.333
C03101=1075.732,354.314,401.441,175.519,30.083,155.332
C03102=1075.725,354.066,401.477,175.515,30.078,155.331
C03103=1075.719,353.819,401.513,175.512,30.072,155.330
C03104=1075.713,353.571,401.549,175.508,30.067,155.329
C03105=1075.707,353.324,401.585,175.505,30.060,155.328
C03106=1075.700,353.077,401.620,175.502,30.055,155.327
C03107=1075.694,352.829,401.656,175.498,30.049,155.326
C03108=1075.688,352.582,401.692,175.495,30.044,155.325
C03109=1075.682,352.334,401.728,175.491,30.038,155.324
C03110=1075.675,352.087,401.763,175.488,30.033,155.323
C03111=1075.669,351.839,401.799,175.484,30.027,155.322
C03112=1075.663,351.593,401.835,175.481,30.022,155.321
C03113=1075.657,351.346,401.870,175.478,30.016,155.320
C03114=1075.651,351.098,401.906,175.474,30.011,155.319
C03115=1075.645,350.850,401.942,175.471,30.006,155.318
C03116=1075.638,350.603,401.977,175.467,30.000,155.317
C03117=1075.632,350.355,402.013,175.464,29.995,155.316
C03118=1075.625,350.108,402.048,175.460,29.989,155.315
C03119=1075.619,349.861,402.084,175.457,29.984,155.314
C03120=1075.613,349.614,402.119,175.454,29.979,155.313
C03121=1075.606,349.366,402.155,175.450,29.973,155.312
C03122=1075.600,349.119,402.190,175.447,29.967,155.311
C03123=1075.594,348.871,402.226,175.443,29.962,155.310
C03124=1075.588,348.624,402.261,175.440,29.956,155.309
C03125=1075.582,348.377,402.297,175.436,29.951,155.308
C03126=1075.575,348.129,402.332,175.433,29.946,155.307
C03127=1075.570,347.881,402.367,175.430,29.940,155.306
C03128=1075.563,347.634,402.402,175.426,29.935,155.305
C03129=1075.557,347.387,402.437,175.423,29.930,155.304
C03130=1075.551,347.139,402.472,175.419,29.924,155.303
C03131=1075.545,346.892,402.508,175.416,29.919,155.302
C03132=1075.538,346.644,402.543,175.412,29.914,155.301
C03133=1075.532,346.397,402.579,175.409,29.908,155.300
C03134=1075.526,346.149,402.613,175.406,29.903,155.299
C03135=1075.520,345.902,402.649,175.402,29.897,155.298
C03136=1075.513,345.654,402.684,175.399,29.892,155.297
C03137=1075.508,345.407,402.719,175.395,29.887,155.296
C03138=1075.502,345.194,402.749,175.393,29.882,155.295
C03139=1075.497,344.981,402.780,175.389,29.878,155.295
C03140=1075.492,344.767,402.810,175.387,29.873,155.294
C03141=1075.486,344.555,402.840,175.384,29.869,155.293
C03142=1075.482,344.341,402.870,175.381,29.864,155.292
C03143=1075.476,344.128,402.901,175.378,29.860,155.291
C03144=1075.470,343.915,402.930,175.375,29.855,155.290
C03145=1075.465,343.702,402.960,175.372,29.851,155.290
C03146=1075.459,343.454,402.996,175.369,29.846,155.289
C03147=1075.453,343.207,403.030,175.365,29.840,155.288
C03148=1075.446,342.959,403.065,175.362,29.835,155.287
C03149=1075.440,342.711,403.099,175.359,29.830,155.286
C03150=1075.434,342.464,403.135,175.355,29.825,155.285
C03151=1075.428,342.216,403.169,175.352,29.819,155.284
C03152=1075.421,341.969,403.204,175.349,29.815,155.283
C03153=1075.415,341.722,403.238,175.346,29.809,155.282
C03154=1075.409,341.474,403.274,175.342,29.804,155.281
C03155=1075.403,341.227,403.308,175.339,29.799,155.280
C03156=1075.397,340.979,403.343,175.336,29.794,155.279
C03157=1075.390,340.731,403.377,175.332,29.789,155.278
C03158=1075.385,340.484,403.412,175.329,29.784,155.277
C03159=1075.378,340.236,403.447,175.325,29.779,155.277
C03160=1075.372,339.989,403.481,175.322,29.773,155.275
C03161=1075.366,339.741,403.516,175.319,29.768,155.275
C03162=1075.360,339.494,403.551,175.316,29.763,155.274
C03163=1075.354,339.246,403.586,175.313,29.758,155.273
C03164=1075.348,338.999,403.620,175.309,29.753,155.272
C03165=1075.342,338.751,403.654,175.306,29.748,155.271
C03166=1075.336,338.504,403.689,175.302,29.743,155.270
C03167=1075.329,338.256,403.723,175.299,29.737,155.269
C03168=1075.324,338.009,403.758,175.296,29.732,155.268
C03169=1075.317,337.761,403.792,175.293,29.727,155.267
C03170=1075.312,337.513,403.826,175.290,29.722,155.266
C03171=1075.305,337.265,403.861,175.286,29.717,155.265
C03172=1075.299,337.019,403.896,175.283,29.713,155.265
C03173=1075.293,336.771,403.930,175.279,29.708,155.264
C03174=1075.287,336.523,403.964,175.276,29.703,155.263
C03175=1075.280,336.275,403.998,175.273,29.698,155.262
C03176=1075.274,336.028,404.032,175.270,29.693,155.261
C03177=1075.268,335.780,404.067,175.267,29.688,155.260
C03178=1075.262,335.533,404.101,175.263,29.683,155.259
C03179=1075.256,335.285,404.135,175.260,29.677,155.258
C03180=1075.250,335.038,404.169,175.256,29.673,155.258
C03181=1075.243,334.791,404.203,175.254,29.668,155.257
C03182=1075.237,334.543,404.237,175.251,29.663,155.256
C03183=1075.231,334.295,404.271,175.247,29.658,155.255
C03184=1075.225,334.047,404.305,175.244,29.653,155.254
C03185=1075.219,333.800,404.339,175.240,29.648,155.253
C03186=1075.213,333.552,404.373,175.238,29.643,155.252
C03187=1075.206,333.304,404.408,175.234,29.638,155.251
C03188=1075.201,333.057,404.442,175.231,29.633,155.250
C03189=1075.194,332.809,404.476,175.228,29.628,155.250
C03190=1075.189,332.561,404.509,175.224,29.624,155.249
C03191=1075.183,332.314,404.543,175.222,29.619,155.248
C03192=1075.176,332.066,404.578,175.218,29.614,155.247
C03193=1075.170,331.819,404.612,175.215,29.609,155.246
C03194=1075.165,331.603,404.640,175.212,29.605,155.245
C03195=1075.160,331.387,404.670,175.209,29.600,155.245
C03196=1075.154,331.171,404.700,175.206,29.596,155.244
C03197=1075.149,330.956,404.729,175.204,29.592,155.243
C03198=1075.143,330.739,404.758,175.201,29.588,155.242
C03199=1075.138,330.525,404.788,175.198,29.584,155.242
C03200=1075.132,330.308,404.817,175.195,29.579,155.241
C03201=1075.127,330.092,404.847,175.193,29.576,155.240
C03202=1075.121,329.845,404.880,175.189,29.571,155.239
C03203=1075.115,329.597,404.914,175.186,29.566,155.239
C03204=1075.108,329.349,404.948,175.183,29.561,155.238
C03205=1075.102,329.101,404.981,175.180,29.556,155.237
C03206=1075.096,328.854,405.014,175.177,29.552,155.236
C03207=1075.089,328.606,405.048,175.173,29.547,155.235
C03208=1075.084,328.359,405.082,175.170,29.542,155.234
C03209=1075.077,328.111,405.115,175.167,29.538,155.234
C03210=1075.071,327.863,405.149,175.164,29.533,155.233
C03211=1075.065,327.615,405.182,175.161,29.528,155.232
C03212=1075.059,327.368,405.215,175.157,29.524,155.231
C03213=1075.052,327.121,405.249,175.155,29.519,155.230
C03214=1075.046,326.872,405.282,175.151,29.514,155.230
C03215=1075.040,326.625,405.316,175.148,29.510,155.229
C03216=1075.034,326.377,405.349,175.145,29.505,155.228
C03217=1075.028,326.129,405.382,175.142,29.500,155.227
C03218=1075.022,325.881,405.416,175.138,29.495,155.226
C03219=1075.015,325.634,405.449,175.135,29.490,155.225
C03220=1075.010,325.386,405.483,175.133,29.486,155.225
C03221=1075.003,325.138,405.515,175.129,29.481,155.224
C03222=1074.997,324.891,405.549,175.126,29.476,155.223
C03223=1074.991,324.644,405.582,175.123,29.472,155.222
C03224=1074.985,324.395,405.616,175.120,29.467,155.221
C03225=1074.979,324.147,405.649,175.116,29.463,155.221
C03226=1074.973,323.899,405.682,175.114,29.458,155.220
C03227=1074.966,323.652,405.715,175.111,29.453,155.219
C03228=1074.961,323.405,405.749,175.107,29.449,155.218
C03229=1074.955,323.157,405.781,175.104,29.444,155.217
C03230=1074.949,322.909,405.815,175.101,29.439,155.216
C03231=1074.943,322.661,405.847,175.098,29.435,155.216
C03232=1074.937,322.414,405.881,175.095,29.430,155.215
C03233=1074.930,322.165,405.914,175.092,29.426,155.214
C03234=1074.924,321.918,405.947,175.089,29.421,155.213
C03235=1074.918,321.670,405.980,175.085,29.416,155.212
C03236=1074.912,321.422,406.013,175.083,29.412,155.212
C03237=1074.907,321.174,406.046,175.079,29.407,155.211
C03238=1074.900,320.927,406.079,175.076,29.402,155.210
C03239=1074.895,320.679,406.112,175.074,29.398,155.209
C03240=1074.888,320.431,406.145,175.070,29.393,155.208
C03241=1074.882,320.184,406.178,175.068,29.389,155.208
C03242=1074.877,319.936,406.211,175.064,29.384,155.207
C03243=1074.870,319.688,406.244,175.061,29.379,155.206
C03244=1074.864,319.440,406.276,175.058,29.375,155.205
C03245=1074.859,319.193,406.310,175.055,29.370,155.205
C03246=1074.852,318.945,406.343,175.052,29.365,155.204
C03247=1074.847,318.697,406.376,175.049,29.361,155.203
C03248=1074.841,318.449,406.408,175.046,29.356,155.202
C03249=1074.835,318.202,406.440,175.043,29.352,155.201
C03250=1074.830,317.983,406.470,175.040,29.348,155.201
C03251=1074.824,317.764,406.499,175.037,29.344,155.200
C03252=1074.819,317.545,406.528,175.035,29.340,155.199
C03253=1074.814,317.326,406.557,175.032,29.336,155.199
C03254=1074.809,317.107,406.586,175.030,29.332,155.198
C03255=1074.803,316.888,406.614,175.026,29.327,155.197
C03256=1074.798,316.668,406.643,175.024,29.323,155.196
C03257=1074.793,316.450,406.672,175.021,29.320,155.196
C03258=1074.788,316.202,406.705,175.018,29.315,155.195
C03259=1074.781,315.954,406.738,175.016,29.311,155.194
C03260=1074.775,315.706,406.770,175.012,29.306,155.193
C03261=1074.770,315.459,406.802,175.010,29.302,155.193
C03262=1074.764,315.211,406.836,175.006,29.297,155.192
C03263=1074.758,314.963,406.868,175.003,29.292,155.191
C03264=1074.752,314.716,406.900,175.001,29.287,155.190
C03265=1074.747,314.467,406.933,174.997,29.283,155.189
C03266=1074.740,314.220,406.965,174.995,29.279,155.189
C03267=1074.734,313.971,406.997,174.991,29.274,155.188
C03268=1074.727,313.724,407.030,174.988,29.270,155.187
C03269=1074.722,313.476,407.062,174.985,29.266,155.187
C03270=1074.716,313.229,407.094,174.982,29.261,155.186
C03271=1074.710,312.981,407.126,174.980,29.257,155.185
C03272=1074.703,312.733,407.159,174.976,29.253,155.184
C03273=1074.697,312.485,407.191,174.974,29.248,155.184
C03274=1074.690,312.237,407.223,174.970,29.244,155.183
C03275=1074.684,311.989,407.255,174.967,29.239,155.182
C03276=1074.678,311.741,407.287,174.964,29.235,155.181
C03277=1074.673,311.494,407.320,174.961,29.231,155.181
C03278=1074.667,311.246,407.352,174.959,29.226,155.180
C03279=1074.661,310.998,407.384,174.955,29.222,155.179
C03280=1074.654,310.750,407.416,174.953,29.218,155.178
C03281=1074.648,310.502,407.448,174.949,29.213,155.178
C03282=1074.642,310.255,407.480,174.946,29.209,155.177
C03283=1074.636,310.007,407.512,174.943,29.204,155.176
C03284=1074.630,309.759,407.544,174.940,29.200,155.176
C03285=1074.623,309.511,407.576,174.937,29.196,155.175
C03286=1074.617,309.263,407.608,174.934,29.191,155.174
C03287=1074.612,309.015,407.639,174.932,29.187,155.173
C03288=1074.606,308.768,407.672,174.928,29.183,155.173
C03289=1074.600,308.519,407.704,174.926,29.178,155.172
C03290=1074.593,308.272,407.735,174.922,29.174,155.171
C03291=1074.587,308.024,407.767,174.919,29.170,155.170
C03292=1074.581,307.776,407.799,174.917,29.165,155.170
C03293=1074.576,307.528,407.831,174.913,29.161,155.169
C03294=1074.569,307.280,407.862,174.911,29.157,155.168
C03295=1074.563,307.033,407.895,174.907,29.153,155.168
C03296=1074.557,306.785,407.927,174.905,29.148,155.167
C03297=1074.552,306.537,407.959,174.901,29.144,155.166
C03298=1074.545,306.289,407.990,174.899,29.140,155.165
C03299=1074.539,306.041,408.022,174.896,29.135,155.165
C03300=1074.534,305.794,408.054,174.893,29.131,155.164
C03301=1074.527,305.546,408.085,174.890,29.127,155.163
C03302=1074.522,305.298,408.117,174.887,29.122,155.162
C03303=1074.516,305.050,408.149,174.884,29.118,155.162
C03304=1074.510,304.802,408.181,174.881,29.114,155.161
C03305=1074.503,304.554,408.212,174.878,29.109,155.160
C03306=1074.499,304.337,408.240,174.876,29.106,155.160
C03307=1074.493,304.120,408.268,174.873,29.102,155.159
C03308=1074.488,303.902,408.295,174.871,29.098,155.158
C03309=1074.483,303.685,408.323,174.868,29.094,155.158
C03310=1074.478,303.467,408.351,174.866,29.091,155.157
C03311=1074.472,303.250,408.379,174.863,29.087,155.157
C03312=1074.467,303.033,408.406,174.861,29.083,155.156
C03313=1074.462,302.815,408.434,174.858,29.079,155.155
C03314=1074.456,302.568,408.465,174.855,29.075,155.155
C03315=1074.450,302.320,408.497,174.852,29.071,155.154
C03316=1074.445,302.072,408.528,174.849,29.066,155.153
C03317=1074.439,301.824,408.560,174.846,29.062,155.152
C03318=1074.433,301.576,408.591,174.843,29.058,155.152
C03319=1074.426,301.328,408.623,174.841,29.053,155.151
C03320=1074.421,301.080,408.654,174.837,29.049,155.150
C03321=1074.415,300.832,408.686,174.835,29.045,155.150
C03322=1074.409,300.585,408.717,174.831,29.041,155.149
C03323=1074.404,300.336,408.748,174.829,29.036,155.148
C03324=1074.397,300.089,408.779,174.826,29.032,155.147
C03325=1074.391,299.840,408.811,174.823,29.028,155.147
C03326=1074.386,299.592,408.842,174.821,29.024,155.146
C03327=1074.380,299.345,408.873,174.817,29.019,155.145
C03328=1074.374,299.097,408.905,174.815,29.015,155.145
C03329=1074.368,298.849,408.936,174.811,29.010,155.144
C03330=1074.362,298.601,408.968,174.809,29.007,155.143
C03331=1074.357,298.353,408.999,174.806,29.002,155.142
C03332=1074.351,298.106,409.030,174.803,28.997,155.142
C03333=1074.346,297.857,409.061,174.801,28.994,155.141
C03334=1074.339,297.609,409.092,174.797,28.989,155.140
C03335=1074.334,297.361,409.123,174.795,28.985,155.140
C03336=1074.328,297.113,409.154,174.792,28.981,155.139
C03337=1074.323,296.865,409.185,174.789,28.976,155.138
C03338=1074.316,296.617,409.217,174.786,28.972,155.138
C03339=1074.310,296.370,409.247,174.783,28.968,155.137
C03340=1074.304,296.121,409.278,174.781,28.964,155.136
C03341=1074.298,295.874,409.310,174.777,28.960,155.135
C03342=1074.292,295.625,409.340,174.775,28.956,155.135
C03343=1074.286,295.377,409.371,174.772,28.952,155.134
C03344=1074.281,295.130,409.402,174.769,28.947,155.133
C03345=1074.274,294.881,409.433,174.766,28.943,155.133
C03346=1074.268,294.633,409.463,174.763,28.939,155.132
C03347=1074.262,294.385,409.495,174.761,28.935,155.131
C03348=1074.257,294.137,409.526,174.758,28.931,155.131
C03349=1074.251,293.889,409.556,174.755,28.927,155.130
C03350=1074.244,293.641,409.587,174.752,28.923,155.129
C03351=1074.238,293.394,409.618,174.749,28.918,155.129
C03352=1074.233,293.146,409.649,174.747,28.914,155.128
C03353=1074.227,292.897,409.679,174.743,28.910,155.127
C03354=1074.221,292.645,409.711,174.741,28.906,155.127
C03355=1074.214,292.393,409.742,174.738,28.902,155.126
C03356=1074.208,292.140,409.773,174.735,28.898,155.125
C03357=1074.203,291.888,409.804,174.733,28.894,155.125
C03358=1074.196,291.640,409.835,174.729,28.889,155.124
C03359=1074.190,291.392,409.866,174.727,28.885,155.123
C03360=1074.185,291.144,409.896,174.724,28.881,155.123
C03361=1074.179,290.896,409.927,174.721,28.877,155.122
C03362=1074.169,290.481,409.978,174.716,28.870,155.121
C03363=1074.159,290.064,410.029,174.712,28.863,155.120
C03364=1074.150,289.649,410.080,174.707,28.856,155.118
C03365=1074.139,289.233,410.131,174.702,28.849,155.117
C03366=1074.133,288.985,410.162,174.700,28.845,155.117
C03367=1074.128,288.737,410.192,174.697,28.841,155.116
C03368=1074.121,288.489,410.223,174.694,28.837,155.115
C03369=1074.115,288.241,410.253,174.691,28.833,155.115
C03370=1074.109,287.993,410.283,174.689,28.829,155.114
C03371=1074.103,287.744,410.313,174.685,28.825,155.113
C03372=1074.098,287.496,410.344,174.683,28.821,155.113
C03373=1074.092,287.248,410.374,174.681,28.817,155.112
C03374=1074.086,287.001,410.404,174.677,28.813,155.111
C03375=1074.079,286.753,410.434,174.675,28.809,155.111
C03376=1074.073,286.505,410.465,174.672,28.805,155.110
C03377=1074.067,286.256,410.495,174.669,28.801,155.109
C03378=1074.062,286.008,410.525,174.667,28.797,155.109
C03379=1074.056,285.760,410.555,174.664,28.793,155.108
C03380=1074.050,285.513,410.586,174.661,28.788,155.107
C03381=1074.044,285.264,410.616,174.658,28.785,155.107
C03382=1074.038,285.016,410.646,174.656,28.781,155.106
C03383=1074.032,284.768,410.676,174.653,28.776,155.105
C03384=1074.026,284.520,410.707,174.650,28.772,155.105
C03385=1074.020,284.272,410.736,174.648,28.768,155.104
C03386=1074.014,284.024,410.766,174.644,28.764,155.103
C03387=1074.008,283.775,410.796,174.642,28.760,155.103
C03388=1074.002,283.527,410.826,174.639,28.756,155.102
C03389=1073.997,283.279,410.857,174.636,28.752,155.102
C03390=1073.991,283.031,410.886,174.634,28.748,155.101
C03391=1073.985,282.783,410.917,174.631,28.744,155.100
C03392=1073.979,282.535,410.946,174.629,28.740,155.100
C03393=1073.973,282.287,410.976,174.625,28.736,155.099
C03394=1073.967,282.039,411.007,174.623,28.732,155.098
C03395=1073.962,281.791,411.036,174.621,28.727,155.097
C03396=1073.956,281.543,411.067,174.617,28.723,155.097
C03397=1073.951,281.295,411.096,174.615,28.719,155.096
C03398=1073.944,281.047,411.126,174.612,28.715,155.096
C03399=1073.938,280.798,411.156,174.610,28.711,155.095
C03400=1073.932,280.550,411.186,174.607,28.707,155.094
C03401=1073.927,280.302,411.216,174.604,28.703,155.094
C03402=1073.920,280.054,411.245,174.602,28.699,155.093
C03403=1073.915,279.806,411.275,174.598,28.695,155.092
C03404=1073.909,279.557,411.305,174.596,28.691,155.092
C03405=1073.903,279.309,411.334,174.593,28.687,155.091
C03406=1073.897,279.061,411.364,174.591,28.683,155.090
C03407=1073.891,278.813,411.393,174.588,28.679,155.090
C03408=1073.885,278.565,411.424,174.585,28.675,155.089
C03409=1073.879,278.317,411.453,174.583,28.671,155.088
C03410=1073.873,278.069,411.482,174.580,28.667,155.088
C03411=1073.868,277.820,411.512,174.577,28.663,155.087
C03412=1073.862,277.573,411.542,174.575,28.659,155.087
C03413=1073.856,277.324,411.571,174.572,28.655,155.086
C03414=1073.845,276.914,411.620,174.567,28.649,155.085
C03415=1073.837,276.504,411.669,174.563,28.642,155.084
C03416=1073.826,276.094,411.718,174.559,28.636,155.083
C03417=1073.817,275.684,411.766,174.554,28.629,155.082
C03418=1073.811,275.436,411.796,174.552,28.625,155.081
C03419=1073.805,275.188,411.825,174.549,28.621,155.080
C03420=1073.799,274.940,411.855,174.547,28.617,155.080
C03421=1073.793,274.692,411.884,174.544,28.613,155.079
C03422=1073.787,274.443,411.914,174.541,28.609,155.078
C03423=1073.781,274.195,411.943,174.539,28.605,155.078
C03424=1073.776,273.947,411.972,174.536,28.601,155.077
C03425=1073.769,273.699,412.001,174.533,28.597,155.077
C03426=1073.764,273.450,412.031,174.530,28.593,155.076
C03427=1073.758,273.202,412.060,174.528,28.589,155.075
C03428=1073.752,272.954,412.090,174.526,28.586,155.075
C03429=1073.746,272.705,412.119,174.522,28.581,155.074
C03430=1073.740,272.458,412.147,174.520,28.577,155.073
C03431=1073.735,272.210,412.177,174.517,28.573,155.073
C03432=1073.728,271.961,412.206,174.515,28.569,155.072
C03433=1073.722,271.713,412.235,174.513,28.566,155.071
C03434=1073.717,271.465,412.265,174.509,28.561,155.071
C03435=1073.710,271.217,412.294,174.507,28.558,155.070
C03436=1073.705,270.968,412.324,174.504,28.554,155.070
C03437=1073.699,270.719,412.352,174.502,28.550,155.069
C03438=1073.693,270.471,412.381,174.500,28.546,155.068
C03439=1073.688,270.224,412.410,174.496,28.542,155.068
C03440=1073.682,269.975,412.439,174.494,28.538,155.067
C03441=1073.675,269.727,412.468,174.491,28.534,155.066
C03442=1073.669,269.479,412.497,174.489,28.530,155.066
C03443=1073.664,269.230,412.526,174.487,28.526,155.065
C03444=1073.658,268.982,412.555,174.483,28.522,155.065
C03445=1073.652,268.735,412.584,174.481,28.518,155.064
C03446=1073.646,268.486,412.613,174.478,28.514,155.063
C03447=1073.641,268.237,412.642,174.476,28.510,155.063
C03448=1073.634,267.989,412.671,174.474,28.506,155.062
C03449=1073.628,267.741,412.700,174.470,28.502,155.061
C03450=1073.622,267.492,412.728,174.468,28.499,155.061
C03451=1073.616,267.245,412.757,174.465,28.495,155.060
C03452=1073.611,266.997,412.787,174.463,28.491,155.060
C03453=1073.605,266.748,412.815,174.461,28.487,155.059
C03454=1073.599,266.500,412.844,174.458,28.483,155.058
C03455=1073.592,266.251,412.873,174.455,28.479,155.058
C03456=1073.587,266.003,412.901,174.452,28.475,155.057
C03457=1073.582,265.755,412.931,174.450,28.471,155.056
C03458=1073.576,265.506,412.959,174.448,28.467,155.056
C03459=1073.569,265.258,412.988,174.445,28.463,155.055
C03460=1073.564,265.010,413.016,174.443,28.459,155.055
C03461=1073.558,264.762,413.045,174.440,28.455,155.054
C03462=1073.552,264.513,413.073,174.437,28.451,155.053
C03463=1073.546,264.266,413.102,174.435,28.448,155.053
C03464=1073.541,264.017,413.131,174.432,28.444,155.052
C03465=1073.535,263.769,413.160,174.430,28.440,155.051
C03466=1073.525,263.362,413.206,174.426,28.434,155.050
C03467=1073.515,262.955,413.252,174.422,28.427,155.049
C03468=1073.505,262.549,413.299,174.417,28.421,155.048
C03469=1073.495,262.142,413.346,174.413,28.415,155.047
C03470=1073.489,261.893,413.375,174.410,28.411,155.047
C03471=1073.484,261.645,413.403,174.408,28.407,155.046
C03472=1073.477,261.397,413.432,174.406,28.403,155.046
C03473=1073.471,261.149,413.459,174.403,28.399,155.045
C03474=1073.465,260.900,413.488,174.400,28.395,155.044
C03475=1073.459,260.652,413.516,174.397,28.392,155.044
C03476=1073.453,260.404,413.545,174.395,28.388,155.043
C03477=1073.447,260.155,413.573,174.393,28.384,155.043
C03478=1073.442,259.907,413.601,174.390,28.380,155.042
C03479=1073.435,259.658,413.629,174.388,28.376,155.041
C03480=1073.429,259.410,413.658,174.385,28.372,155.041
C03481=1073.423,259.162,413.686,174.383,28.368,155.040
C03482=1073.418,258.913,413.714,174.380,28.364,155.040
C03483=1073.412,258.665,413.742,174.377,28.360,155.039
C03484=1073.406,258.417,413.770,174.375,28.356,155.038
C03485=1073.399,258.169,413.799,174.373,28.352,155.038
C03486=1073.393,257.920,413.827,174.370,28.349,155.037
C03487=1073.388,257.672,413.855,174.368,28.345,155.037
C03488=1073.382,257.423,413.883,174.365,28.341,155.036
C03489=1073.375,257.175,413.911,174.363,28.338,155.035
C03490=1073.370,256.927,413.939,174.360,28.334,155.035
C03491=1073.364,256.678,413.967,174.358,28.330,155.034
C03492=1073.359,256.430,413.995,174.355,28.325,155.033
C03493=1073.352,256.182,414.023,174.352,28.322,155.033
C03494=1073.346,255.933,414.051,174.350,28.318,155.032
C03495=1073.341,255.685,414.079,174.348,28.314,155.032
C03496=1073.335,255.436,414.108,174.345,28.310,155.031
C03497=1073.329,255.188,414.135,174.343,28.307,155.030
C03498=1073.323,254.940,414.163,174.340,28.303,155.030
C03499=1073.318,254.691,414.191,174.338,28.299,155.029
C03500=1073.312,254.443,414.220,174.336,28.295,155.028
C03501=1073.306,254.195,414.247,174.333,28.291,155.028
C03502=1073.300,253.946,414.275,174.331,28.287,155.027
C03503=1073.294,253.698,414.303,174.328,28.283,155.027
C03504=1073.288,253.449,414.332,174.325,28.279,155.026
C03505=1073.282,253.201,414.359,174.323,28.275,155.025
C03506=1073.276,252.953,414.387,174.320,28.271,155.025
C03507=1073.271,252.704,414.415,174.318,28.267,155.024
C03508=1073.265,252.456,414.442,174.316,28.263,155.024
C03509=1073.259,252.208,414.470,174.313,28.259,155.023
C03510=1073.253,251.959,414.499,174.311,28.255,155.022
C03511=1073.248,251.711,414.527,174.308,28.252,155.022
C03512=1073.241,251.463,414.554,174.306,28.248,155.021
C03513=1073.236,251.214,414.582,174.304,28.244,155.020
C03514=1073.230,250.965,414.610,174.301,28.240,155.020
C03515=1073.224,250.717,414.637,174.299,28.236,155.019
C03516=1073.218,250.469,414.666,174.297,28.232,155.019
C03517=1073.213,250.220,414.693,174.294,28.228,155.018
C03518=1073.203,249.811,414.738,174.290,28.222,155.017
C03519=1073.194,249.402,414.784,174.286,28.215,155.016
C03520=1073.185,248.992,414.829,174.282,28.209,155.015
C03521=1073.175,248.583,414.875,174.278,28.202,155.014
C03522=1073.170,248.335,414.903,174.276,28.198,155.013
C03523=1073.164,248.086,414.930,174.274,28.195,155.013
C03524=1073.158,247.838,414.958,174.271,28.191,155.012
C03525=1073.153,247.590,414.986,174.269,28.187,155.011
C03526=1073.147,247.341,415.013,174.267,28.183,155.011
C03527=1073.141,247.093,415.041,174.264,28.179,155.010
C03528=1073.135,246.844,415.068,174.262,28.175,155.009
C03529=1073.130,246.596,415.096,174.259,28.171,155.009
C03530=1073.123,246.347,415.123,174.257,28.167,155.008
C03531=1073.118,246.099,415.151,174.254,28.163,155.008
C03532=1073.112,245.850,415.178,174.251,28.159,155.007
C03533=1073.105,245.602,415.205,174.249,28.156,155.007
C03534=1073.100,245.354,415.232,174.247,28.151,155.006
C03535=1073.094,245.105,415.260,174.244,28.147,155.005
C03536=1073.089,244.856,415.287,174.242,28.143,155.005
C03537=1073.083,244.608,415.314,174.240,28.140,155.004
C03538=1073.077,244.359,415.342,174.237,28.136,155.003
C03539=1073.071,244.111,415.369,174.235,28.132,155.003
C03540=1073.065,243.863,415.396,174.233,28.128,155.002
C03541=1073.060,243.615,415.423,174.230,28.124,155.002
C03542=1073.054,243.366,415.450,174.228,28.120,155.001
C03543=1073.048,243.118,415.478,174.225,28.116,155.000
C03544=1073.043,242.869,415.505,174.223,28.112,155.000
C03545=1073.036,242.620,415.532,174.221,28.108,154.999
C03546=1073.030,242.372,415.559,174.218,28.105,154.999
C03547=1073.025,242.124,415.587,174.216,28.101,154.998
C03548=1073.019,241.875,415.614,174.214,28.097,154.997
C03549=1073.013,241.626,415.640,174.211,28.093,154.997
C03550=1073.007,241.378,415.668,174.210,28.090,154.996
C03551=1073.001,241.130,415.694,174.207,28.086,154.995
C03552=1072.996,240.881,415.722,174.205,28.082,154.995
C03553=1072.990,240.632,415.749,174.203,28.078,154.994
C03554=1072.984,240.384,415.775,174.200,28.074,154.994
C03555=1072.977,240.136,415.803,174.198,28.070,154.993
C03556=1072.972,239.887,415.830,174.196,28.067,154.992
C03557=1072.966,239.639,415.857,174.193,28.063,154.992
C03558=1072.961,239.390,415.883,174.191,28.059,154.991
C03559=1072.954,239.141,415.910,174.189,28.055,154.991
C03560=1072.949,238.893,415.937,174.186,28.051,154.990
C03561=1072.943,238.644,415.964,174.184,28.047,154.989
C03562=1072.937,238.397,415.991,174.182,28.043,154.989
C03563=1072.930,238.148,416.018,174.179,28.039,154.988
C03564=1072.925,237.899,416.045,174.177,28.035,154.988
C03565=1072.919,237.651,416.071,174.174,28.031,154.987
C03566=1072.914,237.402,416.099,174.172,28.027,154.986
C03567=1072.908,237.154,416.125,174.170,28.024,154.986
C03568=1072.902,236.905,416.152,174.167,28.020,154.985
C03569=1072.896,236.656,416.179,174.165,28.016,154.984
C03570=1072.886,236.241,416.223,174.161,28.010,154.984
C03571=1072.876,235.825,416.268,174.157,28.003,154.982
C03572=1072.867,235.409,416.313,174.153,27.996,154.981
C03573=1072.858,234.993,416.358,174.149,27.990,154.980
C03574=1072.851,234.744,416.385,174.148,27.986,154.980
C03575=1072.845,234.496,416.411,174.146,27.982,154.979
C03576=1072.840,234.248,416.438,174.143,27.978,154.978
C03577=1072.834,233.999,416.464,174.141,27.975,154.978
C03578=1072.828,233.750,416.490,174.139,27.971,154.977
C03579=1072.823,233.502,416.517,174.136,27.967,154.977
C03580=1072.817,233.254,416.544,174.134,27.963,154.976
C03581=1072.811,233.005,416.570,174.132,27.959,154.976
C03582=1072.805,232.756,416.597,174.129,27.955,154.975
C03583=1072.799,232.507,416.623,174.127,27.951,154.974
C03584=1072.793,232.259,416.650,174.125,27.947,154.974
C03585=1072.787,232.011,416.676,174.122,27.944,154.973
C03586=1072.781,231.762,416.703,174.120,27.939,154.972
C03587=1072.776,231.513,416.729,174.119,27.936,154.972
C03588=1072.770,231.265,416.755,174.116,27.932,154.971
C03589=1072.764,231.017,416.782,174.114,27.928,154.971
C03590=1072.759,230.768,416.808,174.111,27.924,154.970
C03591=1072.753,230.519,416.834,174.109,27.920,154.969
C03592=1072.747,230.271,416.861,174.107,27.916,154.969
C03593=1072.742,230.022,416.887,174.104,27.913,154.968
C03594=1072.735,229.774,416.913,174.102,27.908,154.968
C03595=1072.729,229.526,416.940,174.100,27.904,154.967
C03596=1072.723,229.276,416.966,174.098,27.900,154.966
C03597=1072.718,229.028,416.993,174.096,27.897,154.966
C03598=1072.711,228.779,417.018,174.094,27.893,154.965
C03599=1072.706,228.531,417.045,174.091,27.889,154.964
C03600=1072.700,228.282,417.071,174.089,27.886,154.964
C03601=1072.694,228.034,417.097,174.087,27.882,154.963
C03602=1072.688,227.785,417.123,174.084,27.877,154.963
C03603=1072.682,227.536,417.149,174.082,27.874,154.962
C03604=1072.677,227.288,417.176,174.080,27.870,154.961
C03605=1072.670,227.039,417.201,174.077,27.866,154.961
C03606=1072.665,226.791,417.228,174.076,27.862,154.960
C03607=1072.659,226.542,417.254,174.074,27.859,154.960
C03608=1072.653,226.294,417.280,174.071,27.855,154.959
C03609=1072.647,226.045,417.306,174.069,27.850,154.958
C03610=1072.642,225.796,417.332,174.067,27.846,154.958
C03611=1072.635,225.548,417.358,174.064,27.843,154.957
C03612=1072.630,225.299,417.384,174.062,27.839,154.957
C03613=1072.624,225.050,417.410,174.060,27.835,154.956
C03614=1072.618,224.802,417.436,174.058,27.831,154.955
C03615=1072.612,224.553,417.462,174.056,27.827,154.955
C03616=1072.606,224.304,417.488,174.054,27.823,154.954
C03617=1072.600,224.056,417.514,174.051,27.819,154.954
C03618=1072.595,223.808,417.540,174.049,27.815,154.953
C03619=1072.590,223.559,417.566,174.047,27.812,154.952
C03620=1072.583,223.310,417.591,174.044,27.808,154.952
C03621=1072.578,223.061,417.617,174.043,27.804,154.951
C03622=1072.572,222.850,417.639,174.041,27.800,154.951
C03623=1072.568,222.638,417.662,174.039,27.797,154.950
C03624=1072.563,222.426,417.683,174.037,27.794,154.949
C03625=1072.558,222.213,417.706,174.035,27.790,154.949
C03626=1072.553,222.002,417.728,174.033,27.787,154.948
C03627=1072.548,221.790,417.750,174.032,27.784,154.948
C03628=1072.543,221.577,417.772,174.030,27.780,154.947
C03629=1072.538,221.365,417.793,174.028,27.777,154.947
C03630=1072.533,221.116,417.819,174.025,27.773,154.946
C03631=1072.526,220.868,417.845,174.023,27.769,154.946
